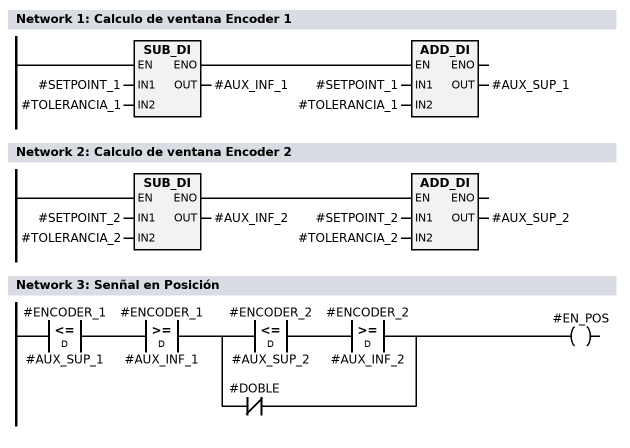
[picture p81: Controlador Posiciones networks 1-3]
NETWORK
TITLE = Calculo de ventana Encoder 1
      A(;
      L     #SETPOINT_1;
      L     #TOLERANCIA_1;
      -D;
      T     #AUX_INF_1;
      AN    OV;
      SAVE;
      CLR;
      A     BR;
      );
      JNB   _001;
      L     #SETPOINT_1;
      L     #TOLERANCIA_1;
      +D;
      T     #AUX_SUP_1;
_001: NOP   0;
NETWORK
TITLE = Calculo de ventana Encoder 2
      A(;
      L     #SETPOINT_2;
      L     #TOLERANCIA_2;
      -D;
      T     #AUX_INF_2;
      AN    OV;
      SAVE;
      CLR;
      A     BR;
      );
      JNB   _002;
      L     #SETPOINT_2;
      L     #TOLERANCIA_2;
      +D;
      T     #AUX_SUP_2;
_002: NOP   0;
NETWORK
TITLE = Senñal en Posición
      A(;
      L     #ENCODER_1;
      L     #AUX_SUP_1;
      <=D;
      );
      A(;
      L     #ENCODER_1;
      L     #AUX_INF_1;
      >=D;
      );
      A(;
      A(;
      L     #ENCODER_2;
      L     #AUX_SUP_2;
      <=D;
      );
      A(;
      L     #ENCODER_2;
      L     #AUX_INF_2;
      >=D;
      );
      ON    #DOBLE;
      );
      =     #EN_POS;
END_FUNCTION

FUNCTION "Almacenes" : VOID	// FC 15
VERSION : 0.1
VAR_TEMP
  TEMP0 : BOOL ;
  TEMP1 : BOOL ;
  TEMP2 : INT ;
END_VAR
BEGIN
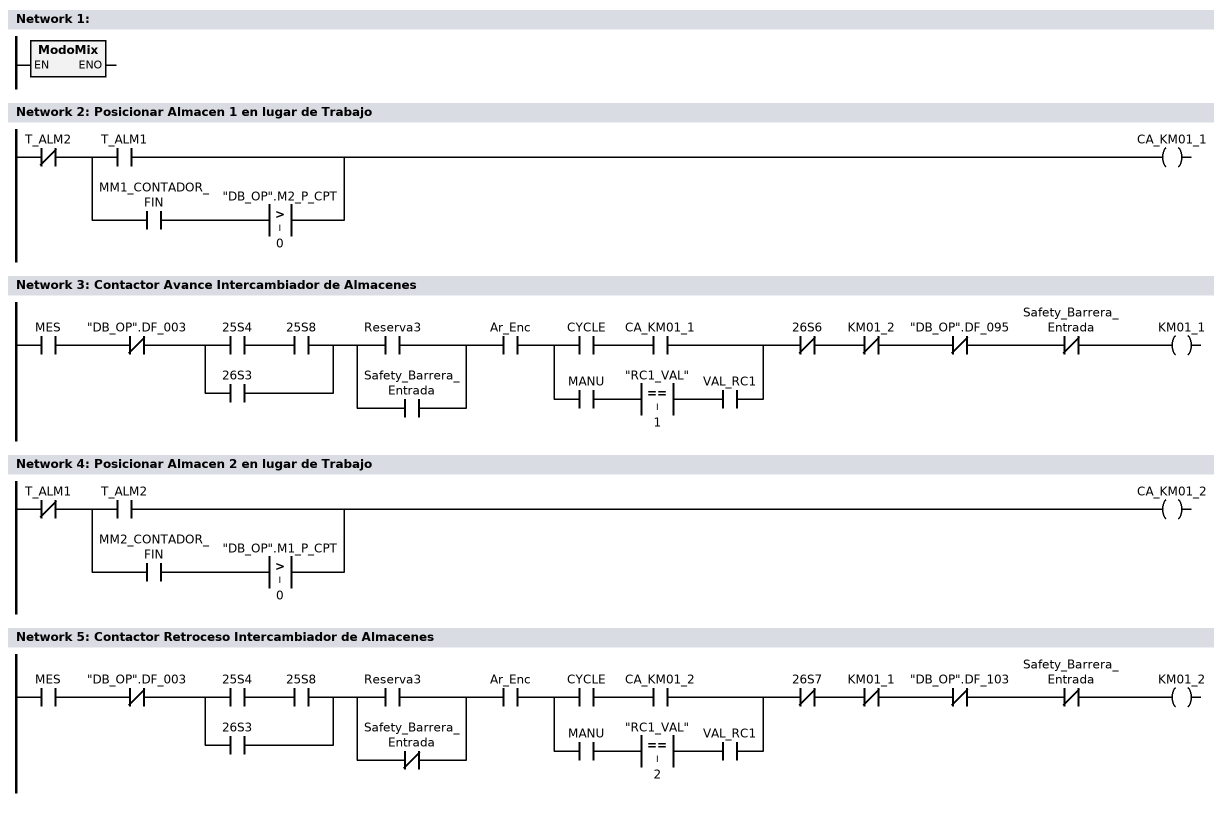
NETWORK
TITLE =
      CALL  "ModoMix";
      NOP   0;
NETWORK
TITLE = Posicionar Almacen 1 en lugar de Trabajo
      AN    "T_ALM2";
      A(;
      O     "T_ALM1";
      O;
      A     "MM1_CONTADOR_FIN";
      A(;
      L     "DB_OP".M2_P_CPT;
      L     0;
      >I;
      );
      );
      =     "CA_KM01_1";
NETWORK
TITLE = Contactor Avance Intercambiador de Almacenes
      A     "MES";
      AN    "DB_OP".DF_003;
      A(;
      A     "25S4";
      A     "25S8";
      O     "26S3";
      );
      A(;
      O     "Reserva3";
      O     "Safety_Barrera_Entrada";
      );
      A     "Ar_Enc";
      A(;
      A     "CYCLE";
      A     "CA_KM01_1";
      O;
      A     "MANU";
      A(;
      L     "RC1_VAL";
      L     1;
      ==I;
      );
      A     "VAL_RC1";
      );
      AN    "26S6";
      AN    "KM01_2";
      AN    "DB_OP".DF_095;
      AN    "Safety_Barrera_Entrada";
      =     "KM01_1";
NETWORK
TITLE = Posicionar Almacen 2 en lugar de Trabajo
      AN    "T_ALM1";
      A(;
      O     "T_ALM2";
      O;
      A     "MM2_CONTADOR_FIN";
      A(;
      L     "DB_OP".M1_P_CPT;
      L     0;
      >I;
      );
      );
      =     "CA_KM01_2";
NETWORK
TITLE = Contactor Retroceso Intercambiador de Almacenes
      A     "MES";
      AN    "DB_OP".DF_003;
      A(;
      A     "25S4";
      A     "25S8";
      O     "26S3";
      );
      A(;
      O     "Reserva3";
      ON    "Safety_Barrera_Entrada";
      );
      A     "Ar_Enc";
      A(;
      A     "CYCLE";
      A     "CA_KM01_2";
      O;
      A     "MANU";
      A(;
      L     "RC1_VAL";
      L     2;
      ==I;
      );
      A     "VAL_RC1";
      );
      AN    "26S7";
      AN    "KM01_1";
      AN    "DB_OP".DF_103;
      AN    "Safety_Barrera_Entrada";
      =     "KM01_2";
END_FUNCTION

FUNCTION "Registro_pos_Plegador" : VOID	// FC 17
TITLE = Registro de posiciones del Plegador
//para verificar el posicionamiento desde el panel
NAME : eProC
VERSION : 0.1
BEGIN
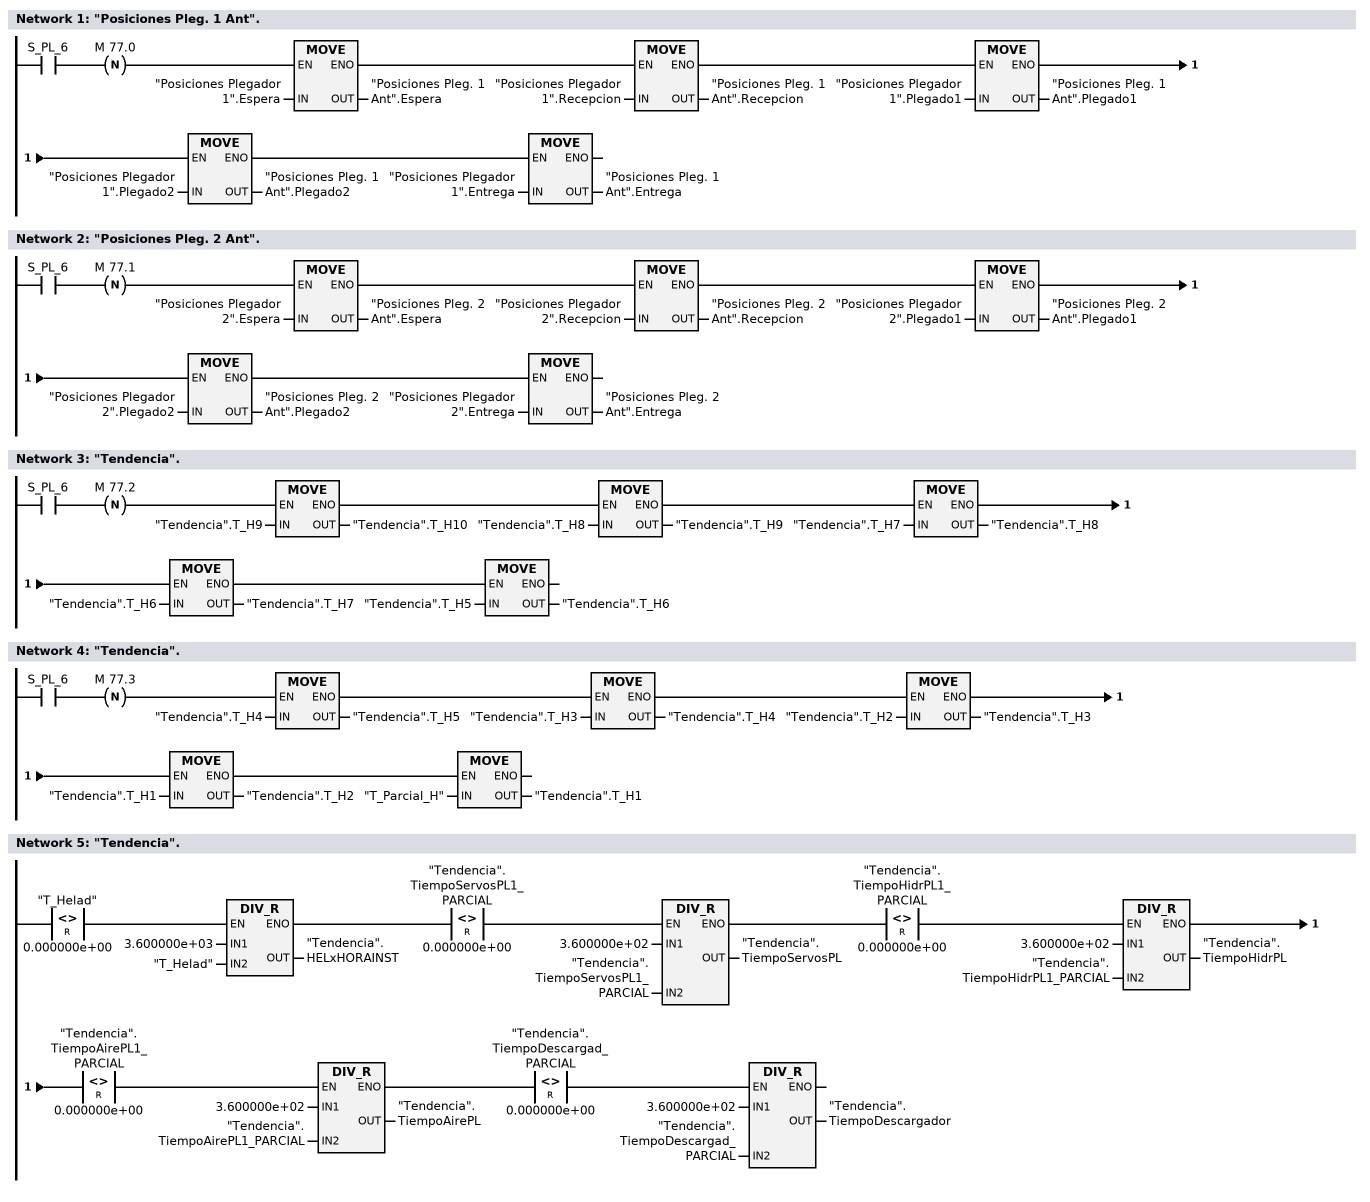
NETWORK
TITLE = "Posiciones Pleg. 1 Ant".
      A(;
      A(;
      A(;
      A(;
      A     "S_PL_6";
      FN    M 77.0;
      JNB   _001;
      L     "Posiciones Plegador 1".Espera;
      T     "Posiciones Pleg. 1 Ant".Espera;
      SET;
      SAVE;
      CLR;
_001: A     BR;
      );
      JNB   _002;
      L     "Posiciones Plegador 1".Recepcion;
      T     "Posiciones Pleg. 1 Ant".Recepcion;
      SET;
      SAVE;
      CLR;
_002: A     BR;
      );
      JNB   _003;
      L     "Posiciones Plegador 1".Plegado1;
      T     "Posiciones Pleg. 1 Ant".Plegado1;
      SET;
      SAVE;
      CLR;
_003: A     BR;
      );
      JNB   _004;
      L     "Posiciones Plegador 1".Plegado2;
      T     "Posiciones Pleg. 1 Ant".Plegado2;
      SET;
      SAVE;
      CLR;
_004: A     BR;
      );
      JNB   _005;
      L     "Posiciones Plegador 1".Entrega;
      T     "Posiciones Pleg. 1 Ant".Entrega;
_005: NOP   0;
NETWORK
TITLE = "Posiciones Pleg. 2 Ant".
      A(;
      A(;
      A(;
      A(;
      A     "S_PL_6";
      FN    M 77.1;
      JNB   _006;
      L     "Posiciones Plegador 2".Espera;
      T     "Posiciones Pleg. 2 Ant".Espera;
      SET;
      SAVE;
      CLR;
_006: A     BR;
      );
      JNB   _007;
      L     "Posiciones Plegador 2".Recepcion;
      T     "Posiciones Pleg. 2 Ant".Recepcion;
      SET;
      SAVE;
      CLR;
_007: A     BR;
      );
      JNB   _008;
      L     "Posiciones Plegador 2".Plegado1;
      T     "Posiciones Pleg. 2 Ant".Plegado1;
      SET;
      SAVE;
      CLR;
_008: A     BR;
      );
      JNB   _009;
      L     "Posiciones Plegador 2".Plegado2;
      T     "Posiciones Pleg. 2 Ant".Plegado2;
      SET;
      SAVE;
      CLR;
_009: A     BR;
      );
      JNB   _00a;
      L     "Posiciones Plegador 2".Entrega;
      T     "Posiciones Pleg. 2 Ant".Entrega;
_00a: NOP   0;
NETWORK
TITLE = "Tendencia".
      A(;
      A(;
      A(;
      A(;
      A     "S_PL_6";
      FN    M 77.2;
      JNB   _00b;
      L     "Tendencia".T_H9;
      T     "Tendencia".T_H10;
      SET;
      SAVE;
      CLR;
_00b: A     BR;
      );
      JNB   _00c;
      L     "Tendencia".T_H8;
      T     "Tendencia".T_H9;
      SET;
      SAVE;
      CLR;
_00c: A     BR;
      );
      JNB   _00d;
      L     "Tendencia".T_H7;
      T     "Tendencia".T_H8;
      SET;
      SAVE;
      CLR;
_00d: A     BR;
      );
      JNB   _00e;
      L     "Tendencia".T_H6;
      T     "Tendencia".T_H7;
      SET;
      SAVE;
      CLR;
_00e: A     BR;
      );
      JNB   _00f;
      L     "Tendencia".T_H5;
      T     "Tendencia".T_H6;
_00f: NOP   0;
NETWORK
TITLE = "Tendencia".
      A(;
      A(;
      A(;
      A(;
      A     "S_PL_6";
      FN    M 77.3;
      JNB   _010;
      L     "Tendencia".T_H4;
      T     "Tendencia".T_H5;
      SET;
      SAVE;
      CLR;
_010: A     BR;
      );
      JNB   _011;
      L     "Tendencia".T_H3;
      T     "Tendencia".T_H4;
      SET;
      SAVE;
      CLR;
_011: A     BR;
      );
      JNB   _012;
      L     "Tendencia".T_H2;
      T     "Tendencia".T_H3;
      SET;
      SAVE;
      CLR;
_012: A     BR;
      );
      JNB   _013;
      L     "Tendencia".T_H1;
      T     "Tendencia".T_H2;
      SET;
      SAVE;
      CLR;
_013: A     BR;
      );
      JNB   _014;
      L     "T_Parcial_H";
      T     "Tendencia".T_H1;
_014: NOP   0;
NETWORK
TITLE = "Tendencia".
      A(;
      A(;
      A(;
      A(;
      A(;
      L     "T_Helad";
      L     0.000000e+00;
      <>R;
      );
      JNB   _015;
      L     3.600000e+03;
      L     "T_Helad";
      /R;
      T     "Tendencia".HELxHORAINST;
      AN    OV;
      SAVE;
      CLR;
_015: A     BR;
      );
      A(;
      L     "Tendencia".TiempoServosPL1_PARCIAL;
      L     0.000000e+00;
      <>R;
      );
      JNB   _016;
      L     3.600000e+02;
      L     "Tendencia".TiempoServosPL1_PARCIAL;
      /R;
      T     "Tendencia".TiempoServosPL;
      AN    OV;
      SAVE;
      CLR;
_016: A     BR;
      );
      A(;
      L     "Tendencia".TiempoHidrPL1_PARCIAL;
      L     0.000000e+00;
      <>R;
      );
      JNB   _017;
      L     3.600000e+02;
      L     "Tendencia".TiempoHidrPL1_PARCIAL;
      /R;
      T     "Tendencia".TiempoHidrPL;
      AN    OV;
      SAVE;
      CLR;
_017: A     BR;
      );
      A(;
      L     "Tendencia".TiempoAirePL1_PARCIAL;
      L     0.000000e+00;
      <>R;
      );
      JNB   _018;
      L     3.600000e+02;
      L     "Tendencia".TiempoAirePL1_PARCIAL;
      /R;
      T     "Tendencia".TiempoAirePL;
      AN    OV;
      SAVE;
      CLR;
_018: A     BR;
      );
      A(;
      L     "Tendencia".TiempoDescargad_PARCIAL;
      L     0.000000e+00;
      <>R;
      );
      JNB   _019;
      L     3.600000e+02;
      L     "Tendencia".TiempoDescargad_PARCIAL;
      /R;
      T     "Tendencia".TiempoDescargador;
_019: NOP   0;
END_FUNCTION

FUNCTION "Registro_pos_Pinza" : VOID	// FC 18
TITLE = Registro de posiciones de la Pinza
//para verificar el posicionamiento desde el panel
NAME : eProC
VERSION : 0.1
BEGIN
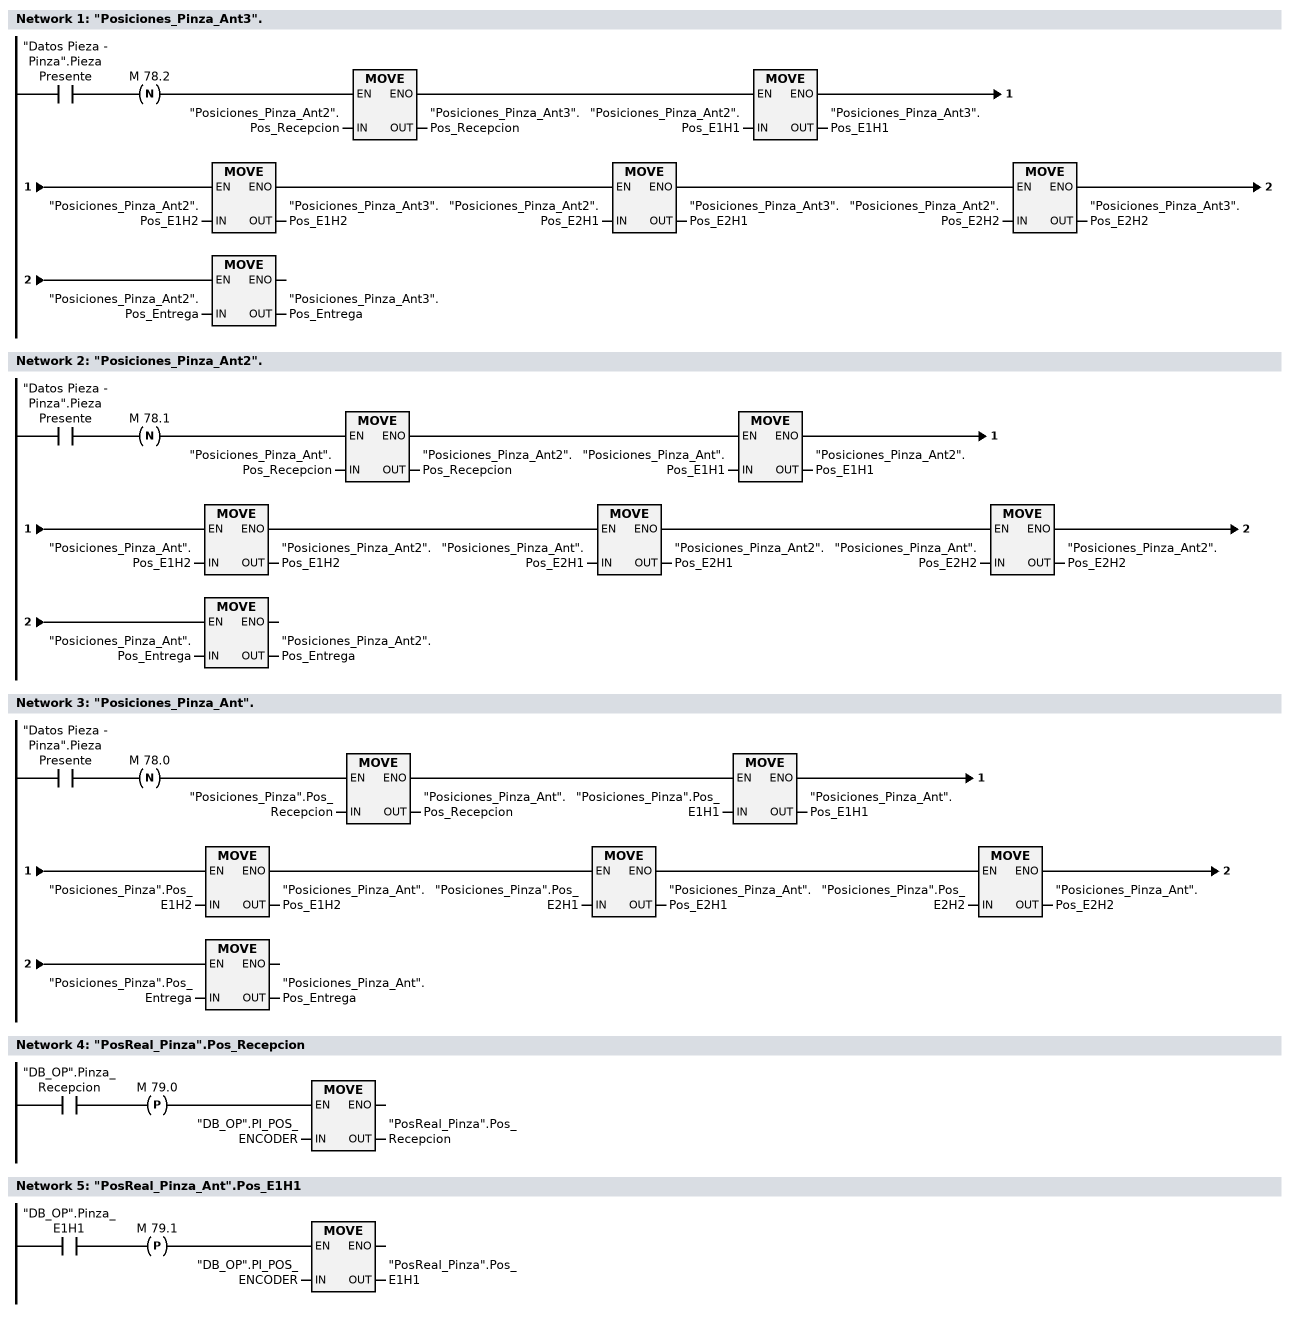
NETWORK
TITLE = "Posiciones_Pinza_Ant3".
      A(;
      A(;
      A(;
      A(;
      A(;
      A     "Datos Pieza - Pinza".PiezaPresente;
      FN    M 78.2;
      JNB   _001;
      L     "Posiciones_Pinza_Ant2".Pos_Recepcion;
      T     "Posiciones_Pinza_Ant3".Pos_Recepcion;
      SET;
      SAVE;
      CLR;
_001: A     BR;
      );
      JNB   _002;
      L     "Posiciones_Pinza_Ant2".Pos_E1H1;
      T     "Posiciones_Pinza_Ant3".Pos_E1H1;
      SET;
      SAVE;
      CLR;
_002: A     BR;
      );
      JNB   _003;
      L     "Posiciones_Pinza_Ant2".Pos_E1H2;
      T     "Posiciones_Pinza_Ant3".Pos_E1H2;
      SET;
      SAVE;
      CLR;
_003: A     BR;
      );
      JNB   _004;
      L     "Posiciones_Pinza_Ant2".Pos_E2H1;
      T     "Posiciones_Pinza_Ant3".Pos_E2H1;
      SET;
      SAVE;
      CLR;
_004: A     BR;
      );
      JNB   _005;
      L     "Posiciones_Pinza_Ant2".Pos_E2H2;
      T     "Posiciones_Pinza_Ant3".Pos_E2H2;
      SET;
      SAVE;
      CLR;
_005: A     BR;
      );
      JNB   _006;
      L     "Posiciones_Pinza_Ant2".Pos_Entrega;
      T     "Posiciones_Pinza_Ant3".Pos_Entrega;
_006: NOP   0;
NETWORK
TITLE = "Posiciones_Pinza_Ant2".
      A(;
      A(;
      A(;
      A(;
      A(;
      A     "Datos Pieza - Pinza".PiezaPresente;
      FN    M 78.1;
      JNB   _007;
      L     "Posiciones_Pinza_Ant".Pos_Recepcion;
      T     "Posiciones_Pinza_Ant2".Pos_Recepcion;
      SET;
      SAVE;
      CLR;
_007: A     BR;
      );
      JNB   _008;
      L     "Posiciones_Pinza_Ant".Pos_E1H1;
      T     "Posiciones_Pinza_Ant2".Pos_E1H1;
      SET;
      SAVE;
      CLR;
_008: A     BR;
      );
      JNB   _009;
      L     "Posiciones_Pinza_Ant".Pos_E1H2;
      T     "Posiciones_Pinza_Ant2".Pos_E1H2;
      SET;
      SAVE;
      CLR;
_009: A     BR;
      );
      JNB   _00a;
      L     "Posiciones_Pinza_Ant".Pos_E2H1;
      T     "Posiciones_Pinza_Ant2".Pos_E2H1;
      SET;
      SAVE;
      CLR;
_00a: A     BR;
      );
      JNB   _00b;
      L     "Posiciones_Pinza_Ant".Pos_E2H2;
      T     "Posiciones_Pinza_Ant2".Pos_E2H2;
      SET;
      SAVE;
      CLR;
_00b: A     BR;
      );
      JNB   _00c;
      L     "Posiciones_Pinza_Ant".Pos_Entrega;
      T     "Posiciones_Pinza_Ant2".Pos_Entrega;
_00c: NOP   0;
NETWORK
TITLE = "Posiciones_Pinza_Ant".
      A(;
      A(;
      A(;
      A(;
      A(;
      A     "Datos Pieza - Pinza".PiezaPresente;
      FN    M 78.0;
      JNB   _00d;
      L     "Posiciones_Pinza".Pos_Recepcion;
      T     "Posiciones_Pinza_Ant".Pos_Recepcion;
      SET;
      SAVE;
      CLR;
_00d: A     BR;
      );
      JNB   _00e;
      L     "Posiciones_Pinza".Pos_E1H1;
      T     "Posiciones_Pinza_Ant".Pos_E1H1;
      SET;
      SAVE;
      CLR;
_00e: A     BR;
      );
      JNB   _00f;
      L     "Posiciones_Pinza".Pos_E1H2;
      T     "Posiciones_Pinza_Ant".Pos_E1H2;
      SET;
      SAVE;
      CLR;
_00f: A     BR;
      );
      JNB   _010;
      L     "Posiciones_Pinza".Pos_E2H1;
      T     "Posiciones_Pinza_Ant".Pos_E2H1;
      SET;
      SAVE;
      CLR;
_010: A     BR;
      );
      JNB   _011;
      L     "Posiciones_Pinza".Pos_E2H2;
      T     "Posiciones_Pinza_Ant".Pos_E2H2;
      SET;
      SAVE;
      CLR;
_011: A     BR;
      );
      JNB   _012;
      L     "Posiciones_Pinza".Pos_Entrega;
      T     "Posiciones_Pinza_Ant".Pos_Entrega;
_012: NOP   0;
NETWORK
TITLE = "PosReal_Pinza".Pos_Recepcion
      A     "DB_OP".Pinza_Recepcion;
      FP    M 79.0;
      JNB   _013;
      L     "DB_OP".PI_POS_ENCODER;
      T     "PosReal_Pinza".Pos_Recepcion;
_013: NOP   0;
NETWORK
TITLE = "PosReal_Pinza_Ant".Pos_E1H1
      A     "DB_OP".Pinza_E1H1;
      FP    M 79.1;
      JNB   _014;
      L     "DB_OP".PI_POS_ENCODER;
      T     "PosReal_Pinza".Pos_E1H1;
_014: NOP   0;
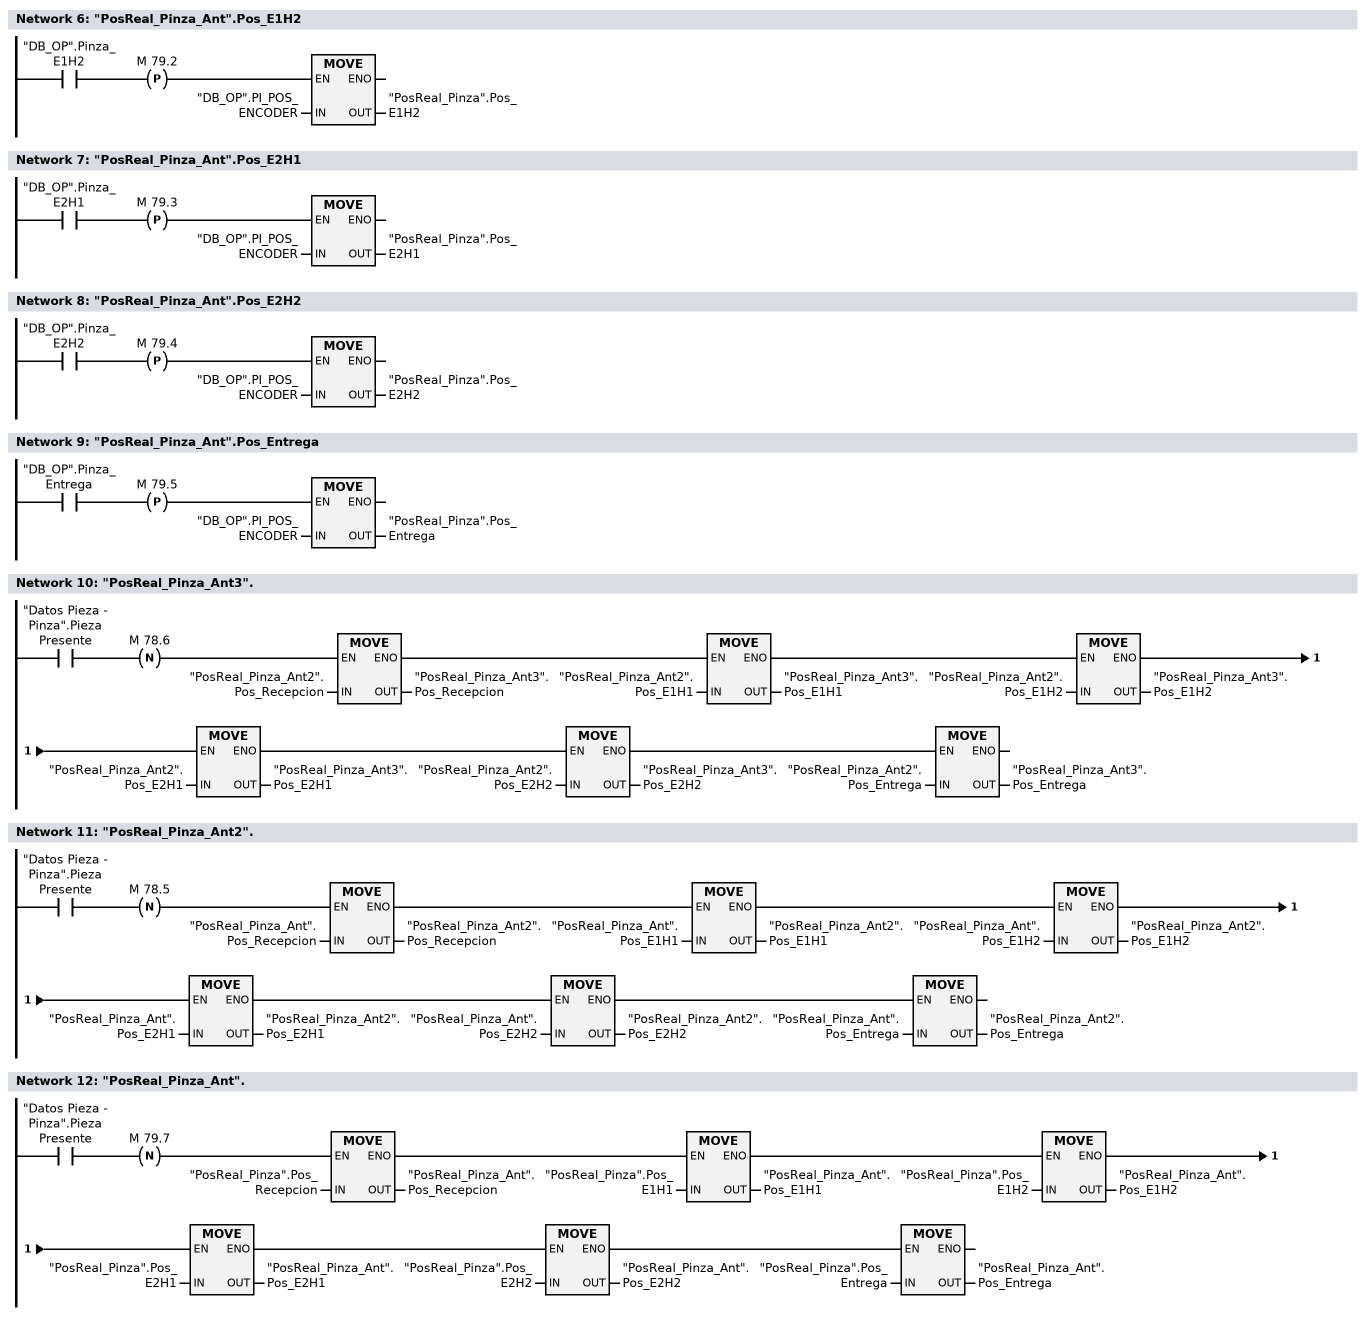
NETWORK
TITLE = "PosReal_Pinza_Ant".Pos_E1H2
      A     "DB_OP".Pinza_E1H2;
      FP    M 79.2;
      JNB   _015;
      L     "DB_OP".PI_POS_ENCODER;
      T     "PosReal_Pinza".Pos_E1H2;
_015: NOP   0;
NETWORK
TITLE = "PosReal_Pinza_Ant".Pos_E2H1
      A     "DB_OP".Pinza_E2H1;
      FP    M 79.3;
      JNB   _016;
      L     "DB_OP".PI_POS_ENCODER;
      T     "PosReal_Pinza".Pos_E2H1;
_016: NOP   0;
NETWORK
TITLE = "PosReal_Pinza_Ant".Pos_E2H2
      A     "DB_OP".Pinza_E2H2;
      FP    M 79.4;
      JNB   _017;
      L     "DB_OP".PI_POS_ENCODER;
      T     "PosReal_Pinza".Pos_E2H2;
_017: NOP   0;
NETWORK
TITLE = "PosReal_Pinza_Ant".Pos_Entrega
      A     "DB_OP".Pinza_Entrega;
      FP    M 79.5;
      JNB   _018;
      L     "DB_OP".PI_POS_ENCODER;
      T     "PosReal_Pinza".Pos_Entrega;
_018: NOP   0;
NETWORK
TITLE = "PosReal_Pinza_Ant3".
      A(;
      A(;
      A(;
      A(;
      A(;
      A     "Datos Pieza - Pinza".PiezaPresente;
      FN    M 78.6;
      JNB   _019;
      L     "PosReal_Pinza_Ant2".Pos_Recepcion;
      T     "PosReal_Pinza_Ant3".Pos_Recepcion;
      SET;
      SAVE;
      CLR;
_019: A     BR;
      );
      JNB   _01a;
      L     "PosReal_Pinza_Ant2".Pos_E1H1;
      T     "PosReal_Pinza_Ant3".Pos_E1H1;
      SET;
      SAVE;
      CLR;
_01a: A     BR;
      );
      JNB   _01b;
      L     "PosReal_Pinza_Ant2".Pos_E1H2;
      T     "PosReal_Pinza_Ant3".Pos_E1H2;
      SET;
      SAVE;
      CLR;
_01b: A     BR;
      );
      JNB   _01c;
      L     "PosReal_Pinza_Ant2".Pos_E2H1;
      T     "PosReal_Pinza_Ant3".Pos_E2H1;
      SET;
      SAVE;
      CLR;
_01c: A     BR;
      );
      JNB   _01d;
      L     "PosReal_Pinza_Ant2".Pos_E2H2;
      T     "PosReal_Pinza_Ant3".Pos_E2H2;
      SET;
      SAVE;
      CLR;
_01d: A     BR;
      );
      JNB   _01e;
      L     "PosReal_Pinza_Ant2".Pos_Entrega;
      T     "PosReal_Pinza_Ant3".Pos_Entrega;
_01e: NOP   0;
NETWORK
TITLE = "PosReal_Pinza_Ant2".
      A(;
      A(;
      A(;
      A(;
      A(;
      A     "Datos Pieza - Pinza".PiezaPresente;
      FN    M 78.5;
      JNB   _01f;
      L     "PosReal_Pinza_Ant".Pos_Recepcion;
      T     "PosReal_Pinza_Ant2".Pos_Recepcion;
      SET;
      SAVE;
      CLR;
_01f: A     BR;
      );
      JNB   _020;
      L     "PosReal_Pinza_Ant".Pos_E1H1;
      T     "PosReal_Pinza_Ant2".Pos_E1H1;
      SET;
      SAVE;
      CLR;
_020: A     BR;
      );
      JNB   _021;
      L     "PosReal_Pinza_Ant".Pos_E1H2;
      T     "PosReal_Pinza_Ant2".Pos_E1H2;
      SET;
      SAVE;
      CLR;
_021: A     BR;
      );
      JNB   _022;
      L     "PosReal_Pinza_Ant".Pos_E2H1;
      T     "PosReal_Pinza_Ant2".Pos_E2H1;
      SET;
      SAVE;
      CLR;
_022: A     BR;
      );
      JNB   _023;
      L     "PosReal_Pinza_Ant".Pos_E2H2;
      T     "PosReal_Pinza_Ant2".Pos_E2H2;
      SET;
      SAVE;
      CLR;
_023: A     BR;
      );
      JNB   _024;
      L     "PosReal_Pinza_Ant".Pos_Entrega;
      T     "PosReal_Pinza_Ant2".Pos_Entrega;
_024: NOP   0;
NETWORK
TITLE = "PosReal_Pinza_Ant".
      A(;
      A(;
      A(;
      A(;
      A(;
      A     "Datos Pieza - Pinza".PiezaPresente;
      FN    M 79.7;
      JNB   _025;
      L     "PosReal_Pinza".Pos_Recepcion;
      T     "PosReal_Pinza_Ant".Pos_Recepcion;
      SET;
      SAVE;
      CLR;
_025: A     BR;
      );
      JNB   _026;
      L     "PosReal_Pinza".Pos_E1H1;
      T     "PosReal_Pinza_Ant".Pos_E1H1;
      SET;
      SAVE;
      CLR;
_026: A     BR;
      );
      JNB   _027;
      L     "PosReal_Pinza".Pos_E1H2;
      T     "PosReal_Pinza_Ant".Pos_E1H2;
      SET;
      SAVE;
      CLR;
_027: A     BR;
      );
      JNB   _028;
      L     "PosReal_Pinza".Pos_E2H1;
      T     "PosReal_Pinza_Ant".Pos_E2H1;
      SET;
      SAVE;
      CLR;
_028: A     BR;
      );
      JNB   _029;
      L     "PosReal_Pinza".Pos_E2H2;
      T     "PosReal_Pinza_Ant".Pos_E2H2;
      SET;
      SAVE;
      CLR;
_029: A     BR;
      );
      JNB   _02a;
      L     "PosReal_Pinza".Pos_Entrega;
      T     "PosReal_Pinza_Ant".Pos_Entrega;
_02a: NOP   0;
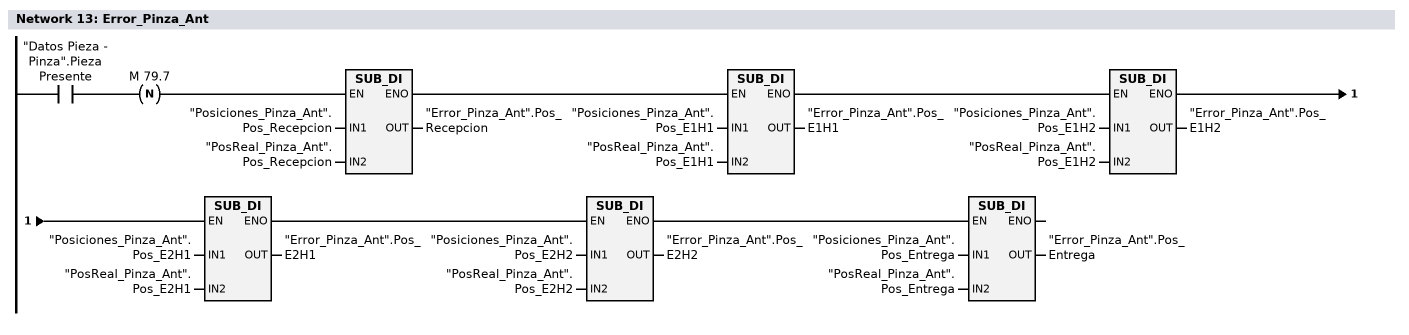
NETWORK
TITLE = Error_Pinza_Ant
      A(;
      A(;
      A(;
      A(;
      A(;
      A     "Datos Pieza - Pinza".PiezaPresente;
      FN    M 79.7;
      JNB   _02b;
      L     "Posiciones_Pinza_Ant".Pos_Recepcion;
      L     "PosReal_Pinza_Ant".Pos_Recepcion;
      -D;
      T     "Error_Pinza_Ant".Pos_Recepcion;
      AN    OV;
      SAVE;
      CLR;
_02b: A     BR;
      );
      JNB   _02c;
      L     "Posiciones_Pinza_Ant".Pos_E1H1;
      L     "PosReal_Pinza_Ant".Pos_E1H1;
      -D;
      T     "Error_Pinza_Ant".Pos_E1H1;
      AN    OV;
      SAVE;
      CLR;
_02c: A     BR;
      );
      JNB   _02d;
      L     "Posiciones_Pinza_Ant".Pos_E1H2;
      L     "PosReal_Pinza_Ant".Pos_E1H2;
      -D;
      T     "Error_Pinza_Ant".Pos_E1H2;
      AN    OV;
      SAVE;
      CLR;
_02d: A     BR;
      );
      JNB   _02e;
      L     "Posiciones_Pinza_Ant".Pos_E2H1;
      L     "PosReal_Pinza_Ant".Pos_E2H1;
      -D;
      T     "Error_Pinza_Ant".Pos_E2H1;
      AN    OV;
      SAVE;
      CLR;
_02e: A     BR;
      );
      JNB   _02f;
      L     "Posiciones_Pinza_Ant".Pos_E2H2;
      L     "PosReal_Pinza_Ant".Pos_E2H2;
      -D;
      T     "Error_Pinza_Ant".Pos_E2H2;
      AN    OV;
      SAVE;
      CLR;
_02f: A     BR;
      );
      JNB   _030;
      L     "Posiciones_Pinza_Ant".Pos_Entrega;
      L     "PosReal_Pinza_Ant".Pos_Entrega;
      -D;
      T     "Error_Pinza_Ant".Pos_Entrega;
_030: NOP   0;
END_FUNCTION

FUNCTION "Araña" : VOID	// FC 20
VERSION : 0.1
VAR_TEMP
  AUX_VELOCIDAD : INT ;	//Auxiliar Consigna de Velocidad
  AUX_CHAPA_COMPLETA : DINT ;
  Arana_A : DINT ;
  Arana_C : DINT ;
  Arana_D : DINT ;
END_VAR
BEGIN
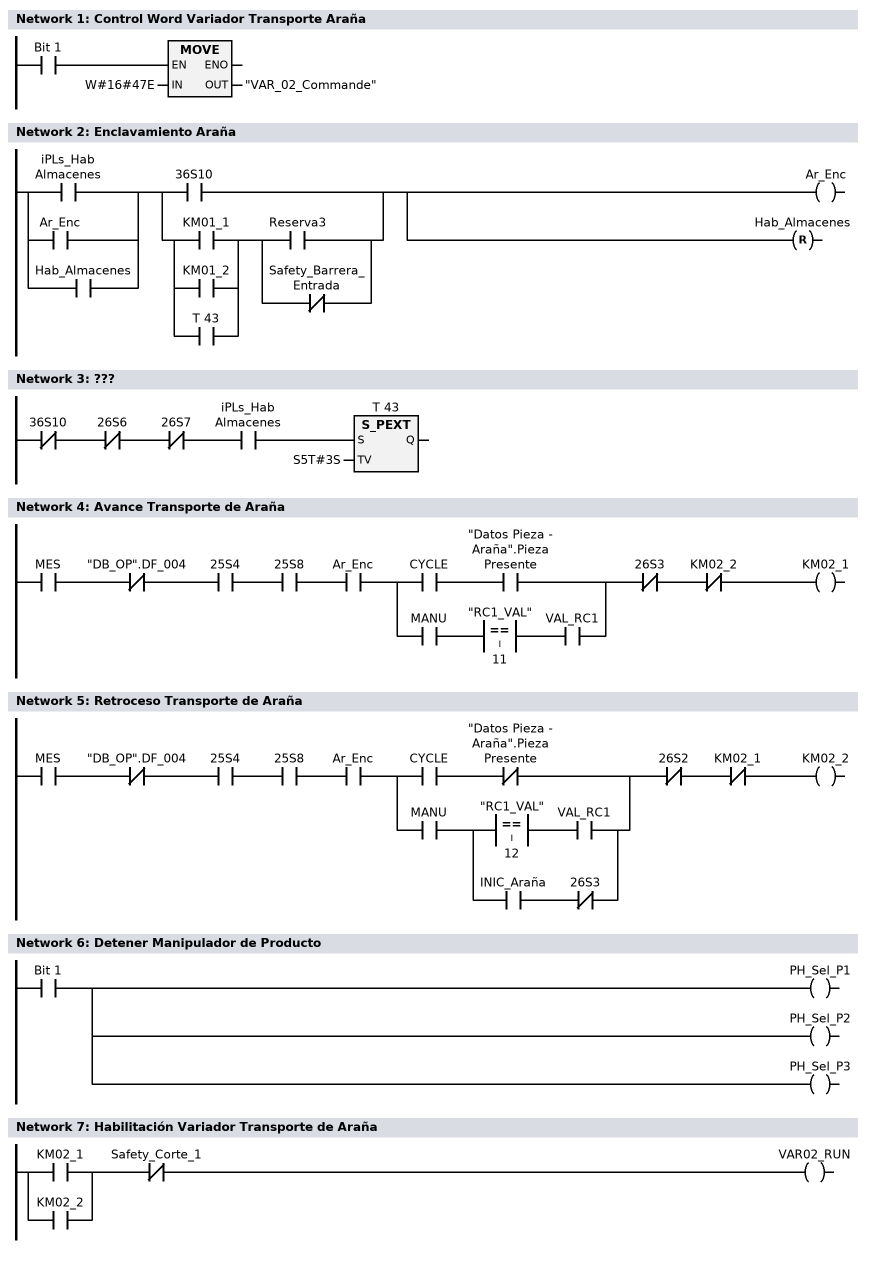
NETWORK
TITLE = Control Word Variador Transporte Araña
      A     "Bit 1";
      JNB   _001;
      L     W#16#47E;
      T     "VAR_02_Commande";
_001: NOP   0;
NETWORK
TITLE = Enclavamiento Araña
      A(;
      O     "iPLs_HabAlmacenes";
      O     "Ar_Enc";
      O     "Hab_Almacenes";
      );
      A(;
      O     "36S10";
      O;
      A(;
      O     "KM01_1";
      O     "KM01_2";
      O     T 43;
      );
      A(;
      O     "Reserva3";
      ON    "Safety_Barrera_Entrada";
      );
      );
      =     "Ar_Enc";
      R     "Hab_Almacenes";
NETWORK
TITLE = ???
      AN    "36S10";
      AN    "26S6";
      AN    "26S7";
      A     "iPLs_HabAlmacenes";
      L     S5T#3S;
      SE    T 43;
      NOP   0;
      NOP   0;
      NOP   0;
      NOP   0;
NETWORK
TITLE = Avance Transporte de Araña
      A     "MES";
      AN    "DB_OP".DF_004;
      A     "25S4";
      A     "25S8";
      A     "Ar_Enc";
      A(;
      A     "CYCLE";
      A     "Datos Pieza - Araña".PiezaPresente;
      O;
      A     "MANU";
      A(;
      L     "RC1_VAL";
      L     11;
      ==I;
      );
      A     "VAL_RC1";
      );
      AN    "26S3";
      AN    "KM02_2";
      =     "KM02_1";
NETWORK
TITLE = Retroceso Transporte de Araña
      A     "MES";
      AN    "DB_OP".DF_004;
      A     "25S4";
      A     "25S8";
      A     "Ar_Enc";
      A(;
      A     "CYCLE";
      AN    "Datos Pieza - Araña".PiezaPresente;
      O;
      A     "MANU";
      A(;
      A(;
      L     "RC1_VAL";
      L     12;
      ==I;
      );
      A     "VAL_RC1";
      O;
      A     "INIC_Araña";
      AN    "26S3";
      );
      );
      AN    "26S2";
      AN    "KM02_1";
      =     "KM02_2";
NETWORK
TITLE = Detener Manipulador de Producto 
      A     "Bit 1";
      =     "PH_Sel_P1";
      =     "PH_Sel_P2";
      =     "PH_Sel_P3";
NETWORK
TITLE = Habilitación Variador Transporte de Araña
      A(;
      O     "KM02_1";
      O     "KM02_2";
      );
      AN    "Safety_Corte_1";
      =     "VAR02_RUN";
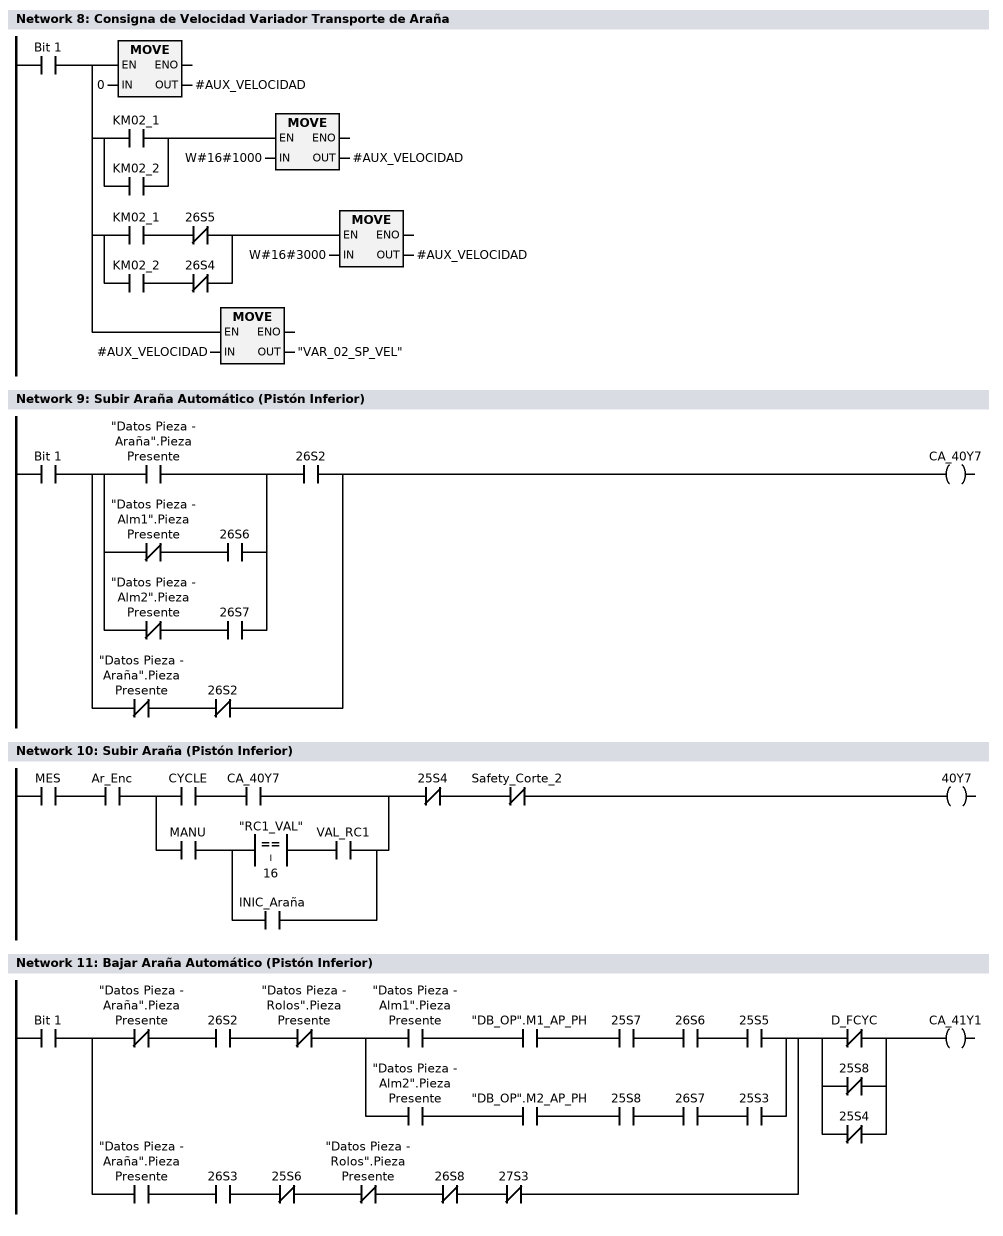
NETWORK
TITLE = Consigna de Velocidad Variador Transporte de Araña
      A     "Bit 1";
      =     L 18.0;
      A     L 18.0;
      JNB   _002;
      L     0;
      T     #AUX_VELOCIDAD;
_002: NOP   0;
      A     L 18.0;
      A(;
      O     "KM02_1";
      O     "KM02_2";
      );
      JNB   _003;
      L     W#16#1000;
      T     #AUX_VELOCIDAD;
_003: NOP   0;
      A     L 18.0;
      A(;
      A     "KM02_1";
      AN    "26S5";
      O;
      A     "KM02_2";
      AN    "26S4";
      );
      JNB   _004;
      L     W#16#3000;
      T     #AUX_VELOCIDAD;
_004: NOP   0;
      A     L 18.0;
      JNB   _005;
      L     #AUX_VELOCIDAD;
      T     "VAR_02_SP_VEL";
_005: NOP   0;
NETWORK
TITLE = Subir Araña Automático (Pistón Inferior)
      A     "Bit 1";
      A(;
      A(;
      O     "Datos Pieza - Araña".PiezaPresente;
      O;
      AN    "Datos Pieza - Alm1".PiezaPresente;
      A     "26S6";
      O;
      AN    "Datos Pieza - Alm2".PiezaPresente;
      A     "26S7";
      );
      A     "26S2";
      O;
      AN    "Datos Pieza - Araña".PiezaPresente;
      AN    "26S2";
      );
      =     "CA_40Y7";
NETWORK
TITLE = Subir Araña (Pistón Inferior)
      A     "MES";
      A     "Ar_Enc";
      A(;
      A     "CYCLE";
      A     "CA_40Y7";
      O;
      A     "MANU";
      A(;
      A(;
      L     "RC1_VAL";
      L     16;
      ==I;
      );
      A     "VAL_RC1";
      O     "INIC_Araña";
      );
      );
      AN    "25S4";
      AN    "Safety_Corte_2";
      =     "40Y7";
NETWORK
TITLE = Bajar Araña Automático (Pistón Inferior)
      A     "Bit 1";
      A(;
      AN    "Datos Pieza - Araña".PiezaPresente;
      A     "26S2";
      AN    "Datos Pieza - Rolos".PiezaPresente;
      A(;
      A     "Datos Pieza - Alm1".PiezaPresente;
      A     "DB_OP".M1_AP_PH;
      A     "25S7";
      A     "26S6";
      A     "25S5";
      O;
      A     "Datos Pieza - Alm2".PiezaPresente;
      A     "DB_OP".M2_AP_PH;
      A     "25S8";
      A     "26S7";
      A     "25S3";
      );
      O;
      A     "Datos Pieza - Araña".PiezaPresente;
      A     "26S3";
      AN    "25S6";
      AN    "Datos Pieza - Rolos".PiezaPresente;
      AN    "26S8";
      AN    "27S3";
      );
      A(;
      ON    "D_FCYC";
      ON    "25S8";
      ON    "25S4";
      );
      =     "CA_41Y1";
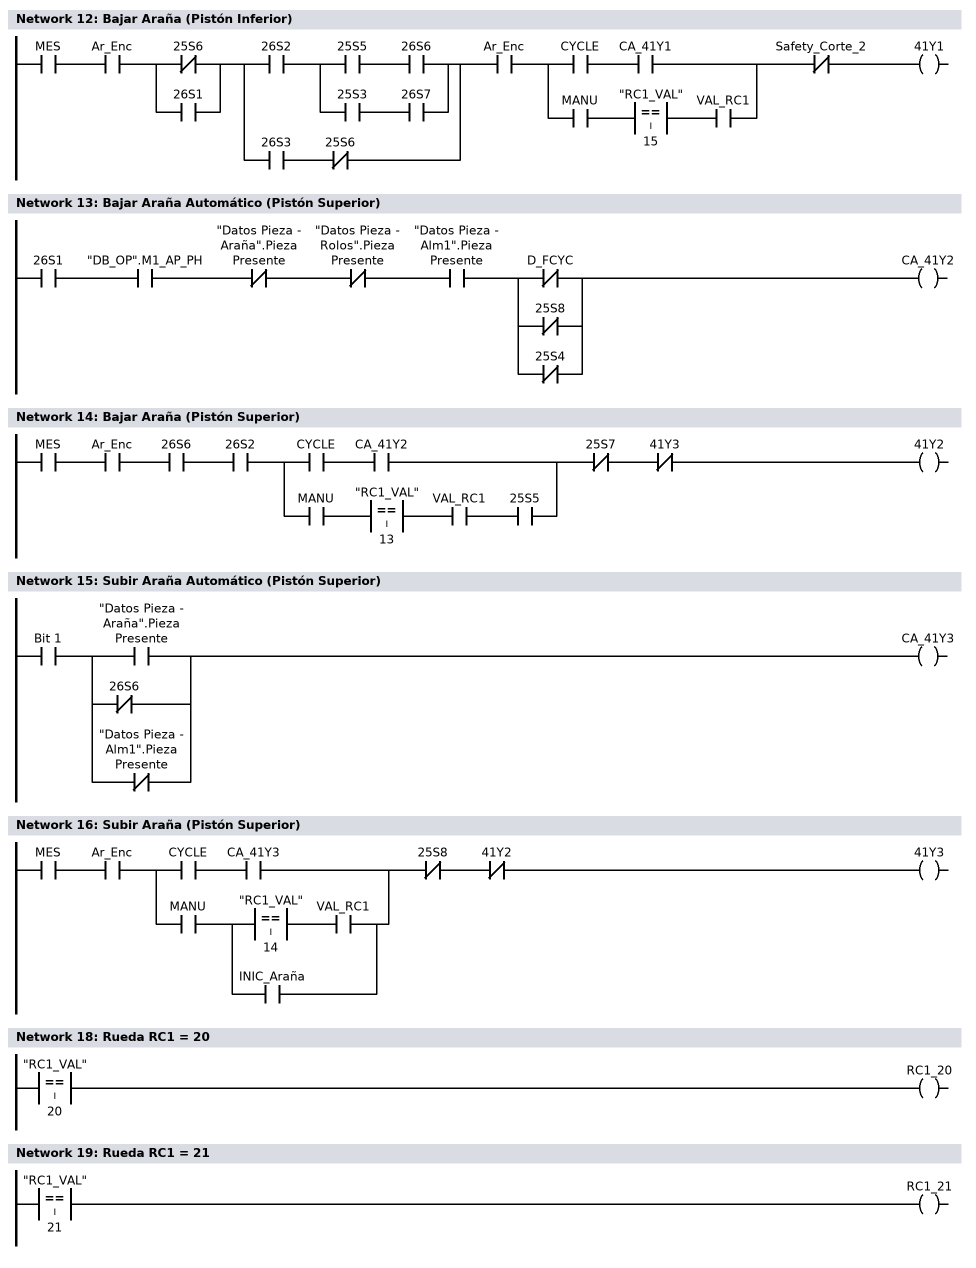
NETWORK
TITLE = Bajar Araña (Pistón Inferior)
      A     "MES";
      A     "Ar_Enc";
      A(;
      ON    "25S6";
      O     "26S1";
      );
      A(;
      A     "26S2";
      A(;
      A     "25S5";
      A     "26S6";
      O;
      A     "25S3";
      A     "26S7";
      );
      O;
      A     "26S3";
      AN    "25S6";
      );
      A     "Ar_Enc";
      A(;
      A     "CYCLE";
      A     "CA_41Y1";
      O;
      A     "MANU";
      A(;
      L     "RC1_VAL";
      L     15;
      ==I;
      );
      A     "VAL_RC1";
      );
      AN    "Safety_Corte_2";
      =     "41Y1";
NETWORK
TITLE = Bajar Araña Automático (Pistón Superior)
      A     "26S1";
      A     "DB_OP".M1_AP_PH;
      AN    "Datos Pieza - Araña".PiezaPresente;
      AN    "Datos Pieza - Rolos".PiezaPresente;
      A     "Datos Pieza - Alm1".PiezaPresente;
      A(;
      ON    "D_FCYC";
      ON    "25S8";
      ON    "25S4";
      );
      =     "CA_41Y2";
NETWORK
TITLE = Bajar Araña (Pistón Superior)
      A     "MES";
      A     "Ar_Enc";
      A     "26S6";
      A     "26S2";
      A(;
      A     "CYCLE";
      A     "CA_41Y2";
      O;
      A     "MANU";
      A(;
      L     "RC1_VAL";
      L     13;
      ==I;
      );
      A     "VAL_RC1";
      A     "25S5";
      );
      AN    "25S7";
      AN    "41Y3";
      =     "41Y2";
NETWORK
TITLE = Subir Araña Automático (Pistón Superior)
      A     "Bit 1";
      A(;
      O     "Datos Pieza - Araña".PiezaPresente;
      ON    "26S6";
      ON    "Datos Pieza - Alm1".PiezaPresente;
      );
      =     "CA_41Y3";
NETWORK
TITLE = Subir Araña (Pistón Superior)
      A     "MES";
      A     "Ar_Enc";
      A(;
      A     "CYCLE";
      A     "CA_41Y3";
      O;
      A     "MANU";
      A(;
      A(;
      L     "RC1_VAL";
      L     14;
      ==I;
      );
      A     "VAL_RC1";
      O     "INIC_Araña";
      );
      );
      AN    "25S8";
      AN    "41Y2";
      =     "41Y3";
NETWORK
TITLE = (COMENTADO EN AWL)
//      U     "MANU"
//      U(    
//      O(    
//      L     "RC1_VAL"
//      L     20
//      ==I   
//      )     
//      O(    
//      L     "RC1_VAL"
//      L     22
//      ==I   
//      )     
//     )     
//      =     #TEMP1
NETWORK
TITLE = Rueda RC1 = 20
      L     "RC1_VAL";
      L     20;
      ==I;
      =     "RC1_20";
NETWORK
TITLE = Rueda RC1 = 21
      L     "RC1_VAL";
      L     21;
      ==I;
      =     "RC1_21";
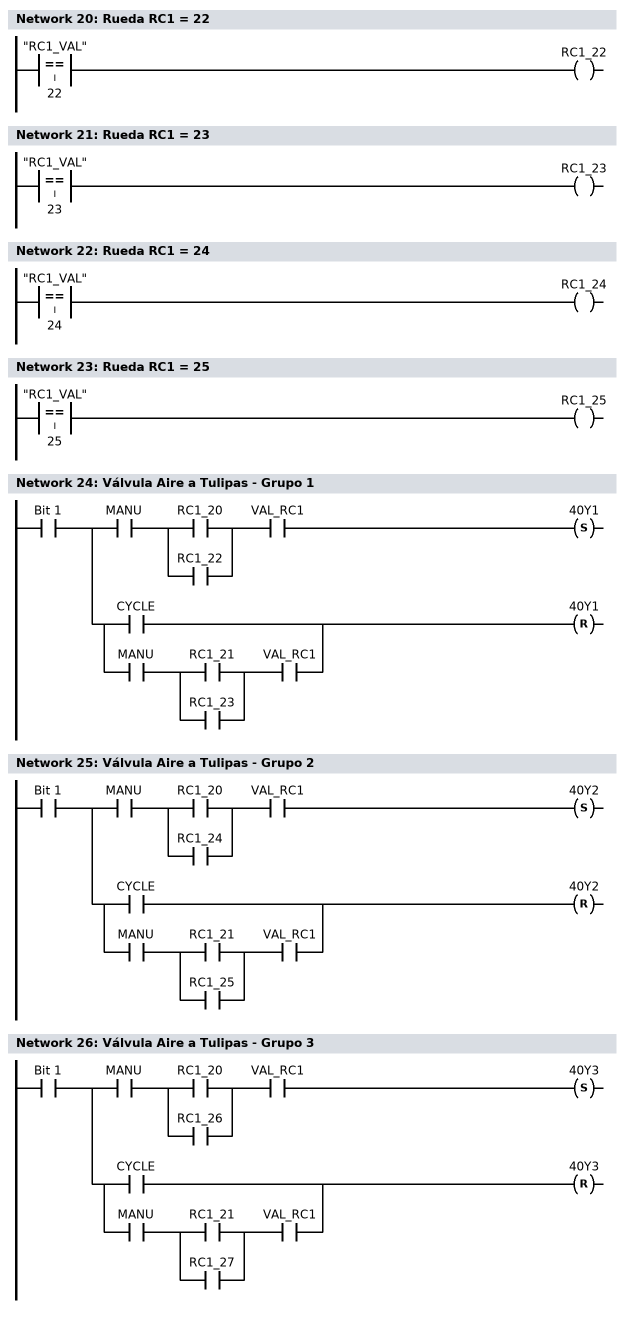
NETWORK
TITLE = Rueda RC1 = 22
      L     "RC1_VAL";
      L     22;
      ==I;
      =     "RC1_22";
NETWORK
TITLE = Rueda RC1 = 23
      L     "RC1_VAL";
      L     23;
      ==I;
      =     "RC1_23";
NETWORK
TITLE = Rueda RC1 = 24
      L     "RC1_VAL";
      L     24;
      ==I;
      =     "RC1_24";
NETWORK
TITLE = Rueda RC1 = 25
      L     "RC1_VAL";
      L     25;
      ==I;
      =     "RC1_25";
NETWORK
TITLE = Válvula Aire a Tulipas - Grupo 1
      A     "Bit 1";
      =     L 18.0;
      A     L 18.0;
      A     "MANU";
      A(;
      O     "RC1_20";
      O     "RC1_22";
      );
      A     "VAL_RC1";
      S     "40Y1";
      A     L 18.0;
      A(;
      O     "CYCLE";
      O;
      A     "MANU";
      A(;
      O     "RC1_21";
      O     "RC1_23";
      );
      A     "VAL_RC1";
      );
      R     "40Y1";
NETWORK
TITLE = Válvula Aire a Tulipas - Grupo 2
      A     "Bit 1";
      =     L 18.0;
      A     L 18.0;
      A     "MANU";
      A(;
      O     "RC1_20";
      O     "RC1_24";
      );
      A     "VAL_RC1";
      S     "40Y2";
      A     L 18.0;
      A(;
      O     "CYCLE";
      O;
      A     "MANU";
      A(;
      O     "RC1_21";
      O     "RC1_25";
      );
      A     "VAL_RC1";
      );
      R     "40Y2";
NETWORK
TITLE = Válvula Aire a Tulipas - Grupo 3
      A     "Bit 1";
      =     L 18.0;
      A     L 18.0;
      A     "MANU";
      A(;
      O     "RC1_20";
      O     "RC1_26";
      );
      A     "VAL_RC1";
      S     "40Y3";
      A     L 18.0;
      A(;
      O     "CYCLE";
      O;
      A     "MANU";
      A(;
      O     "RC1_21";
      O     "RC1_27";
      );
      A     "VAL_RC1";
      );
      R     "40Y3";
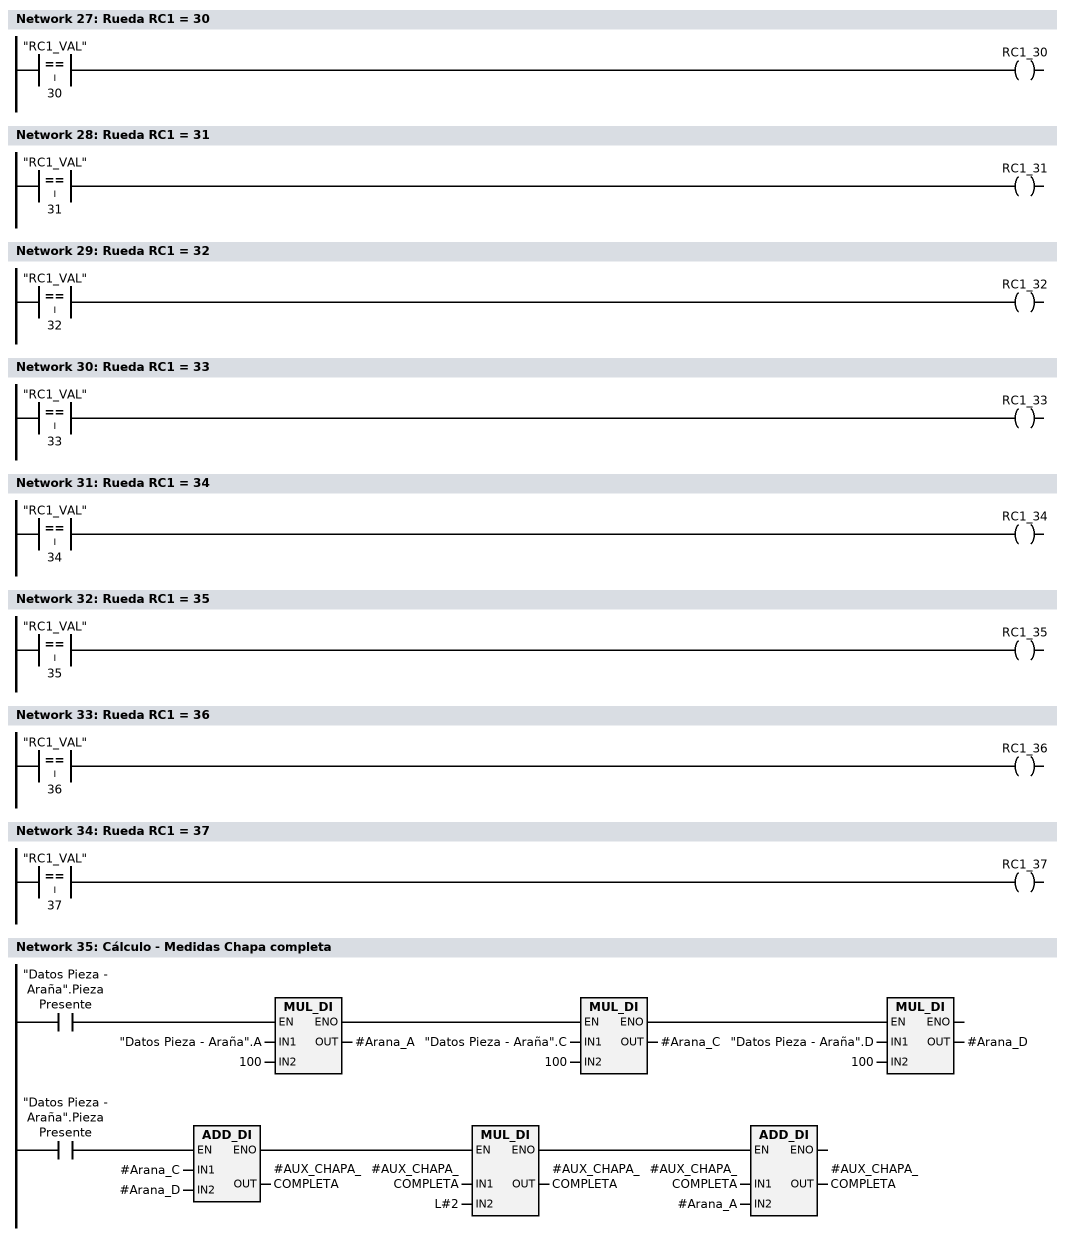
NETWORK
TITLE = Rueda RC1 = 30
      L     "RC1_VAL";
      L     30;
      ==I;
      =     "RC1_30";
NETWORK
TITLE = Rueda RC1 = 31
      L     "RC1_VAL";
      L     31;
      ==I;
      =     "RC1_31";
NETWORK
TITLE = Rueda RC1 = 32
      L     "RC1_VAL";
      L     32;
      ==I;
      =     "RC1_32";
NETWORK
TITLE = Rueda RC1 = 33
      L     "RC1_VAL";
      L     33;
      ==I;
      =     "RC1_33";
NETWORK
TITLE = Rueda RC1 = 34
      L     "RC1_VAL";
      L     34;
      ==I;
      =     "RC1_34";
NETWORK
TITLE = Rueda RC1 = 35
      L     "RC1_VAL";
      L     35;
      ==I;
      =     "RC1_35";
NETWORK
TITLE = Rueda RC1 = 36
      L     "RC1_VAL";
      L     36;
      ==I;
      =     "RC1_36";
NETWORK
TITLE = Rueda RC1 = 37
      L     "RC1_VAL";
      L     37;
      ==I;
      =     "RC1_37";
NETWORK
TITLE = Cálculo - Medidas Chapa completa 
      A     "Datos Pieza - Araña".PiezaPresente;
      =     L 18.0;
      A(;
      A(;
      A     L 18.0;
      JNB   _006;
      L     "Datos Pieza - Araña".A;
      L     100;
      *D;
      T     #Arana_A;
      AN    OV;
      SAVE;
      CLR;
_006: A     BR;
      );
      JNB   _007;
      L     "Datos Pieza - Araña".C;
      L     100;
      *D;
      T     #Arana_C;
      AN    OV;
      SAVE;
      CLR;
_007: A     BR;
      );
      JNB   _008;
      L     "Datos Pieza - Araña".D;
      L     100;
      *D;
      T     #Arana_D;
_008: NOP   0;
      A(;
      A(;
      A     L 18.0;
      JNB   _009;
      L     #Arana_C;
      L     #Arana_D;
      +D;
      T     #AUX_CHAPA_COMPLETA;
      AN    OV;
      SAVE;
      CLR;
_009: A     BR;
      );
      JNB   _00a;
      L     #AUX_CHAPA_COMPLETA;
      L     L#2;
      *D;
      T     #AUX_CHAPA_COMPLETA;
      AN    OV;
      SAVE;
      CLR;
_00a: A     BR;
      );
      JNB   _00b;
      L     #AUX_CHAPA_COMPLETA;
      L     #Arana_A;
      +D;
      T     #AUX_CHAPA_COMPLETA;
_00b: NOP   0;
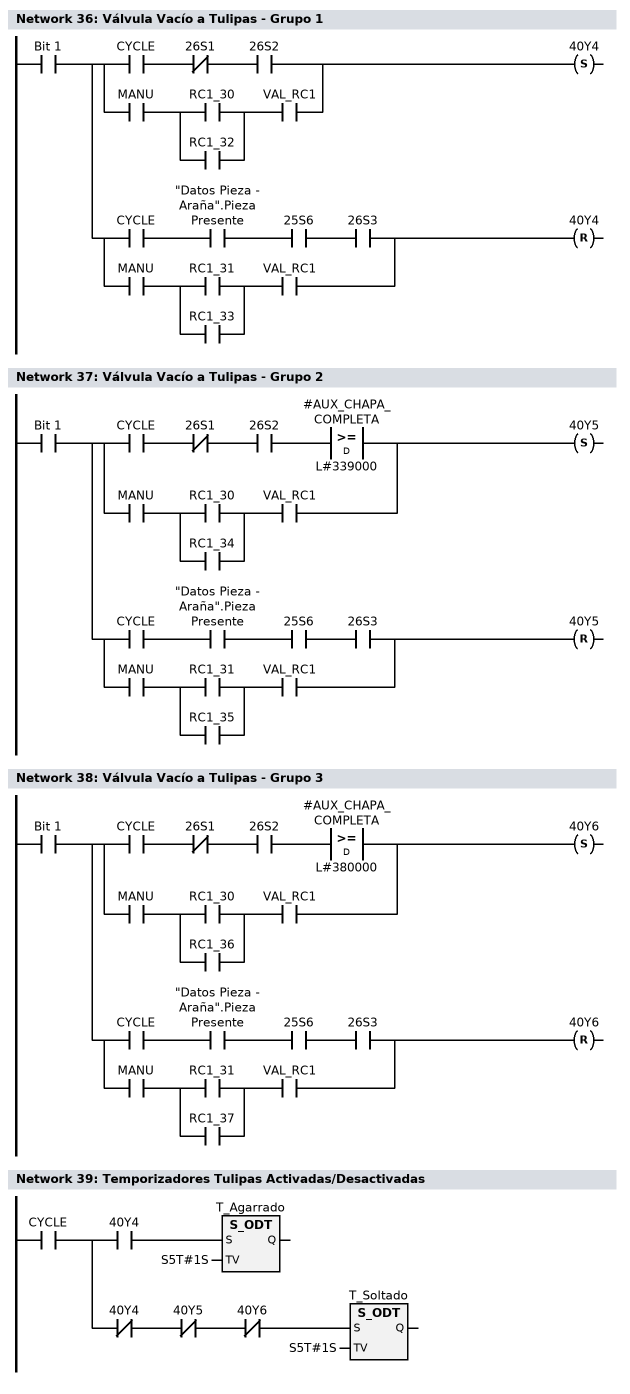
NETWORK
TITLE = Válvula Vacío a Tulipas - Grupo 1
      A     "Bit 1";
      =     L 18.0;
      A     L 18.0;
      A(;
      A     "CYCLE";
      AN    "26S1";
      A     "26S2";
      O;
      A     "MANU";
      A(;
      O     "RC1_30";
      O     "RC1_32";
      );
      A     "VAL_RC1";
      );
      S     "40Y4";
      A     L 18.0;
      A(;
      A     "CYCLE";
      A     "Datos Pieza - Araña".PiezaPresente;
      A     "25S6";
      A     "26S3";
      O;
      A     "MANU";
      A(;
      O     "RC1_31";
      O     "RC1_33";
      );
      A     "VAL_RC1";
      );
      R     "40Y4";
NETWORK
TITLE = Válvula Vacío a Tulipas - Grupo 2
      A     "Bit 1";
      =     L 18.0;
      A     L 18.0;
      A(;
      A     "CYCLE";
      AN    "26S1";
      A     "26S2";
      A(;
      L     #AUX_CHAPA_COMPLETA;
      L     L#339000;
      >=D;
      );
      O;
      A     "MANU";
      A(;
      O     "RC1_30";
      O     "RC1_34";
      );
      A     "VAL_RC1";
      );
      S     "40Y5";
      A     L 18.0;
      A(;
      A     "CYCLE";
      A     "Datos Pieza - Araña".PiezaPresente;
      A     "25S6";
      A     "26S3";
      O;
      A     "MANU";
      A(;
      O     "RC1_31";
      O     "RC1_35";
      );
      A     "VAL_RC1";
      );
      R     "40Y5";
NETWORK
TITLE = Válvula Vacío a Tulipas - Grupo 3
      A     "Bit 1";
      =     L 18.0;
      A     L 18.0;
      A(;
      A     "CYCLE";
      AN    "26S1";
      A     "26S2";
      A(;
      L     #AUX_CHAPA_COMPLETA;
      L     L#380000;
      >=D;
      );
      O;
      A     "MANU";
      A(;
      O     "RC1_30";
      O     "RC1_36";
      );
      A     "VAL_RC1";
      );
      S     "40Y6";
      A     L 18.0;
      A(;
      A     "CYCLE";
      A     "Datos Pieza - Araña".PiezaPresente;
      A     "25S6";
      A     "26S3";
      O;
      A     "MANU";
      A(;
      O     "RC1_31";
      O     "RC1_37";
      );
      A     "VAL_RC1";
      );
      R     "40Y6";
NETWORK
TITLE = Temporizadores Tulipas Activadas/Desactivadas
      A     "CYCLE";
      =     L 18.0;
      A     L 18.0;
      A     "40Y4";
      L     S5T#1S;
      SD    "T_Agarrado";
      NOP   0;
      NOP   0;
      NOP   0;
      NOP   0;
      A     L 18.0;
      AN    "40Y4";
      AN    "40Y5";
      AN    "40Y6";
      L     S5T#1S;
      SD    "T_Soltado";
      NOP   0;
      NOP   0;
      NOP   0;
      NOP   0;
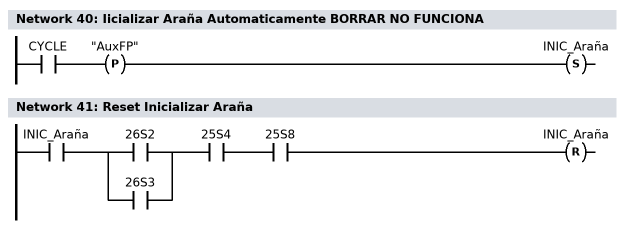
NETWORK
TITLE = Iicializar Araña Automaticamente BORRAR NO FUNCIONA
      A     "CYCLE";
      FP    "AuxFP";
      S     "INIC_Araña";
NETWORK
TITLE = Reset Inicializar Araña
      A     "INIC_Araña";
      A(;
      O     "26S2";
      O     "26S3";
      );
      A     "25S4";
      A     "25S8";
      R     "INIC_Araña";
END_FUNCTION

FUNCTION "Descarga" : VOID	// FC 40
//LUC - 13/08/2020
VERSION : 0.1
VAR_TEMP
  SECU : BOOL ;	//Sécurité mécanique du mouvement
  AUX_SECU : BOOL ;
  NMVT : INT ;	//Numero Mouvement
  M01 : BOOL ;
  FEN_P : DINT ;
  FEN_N : DINT ;
END_VAR
BEGIN
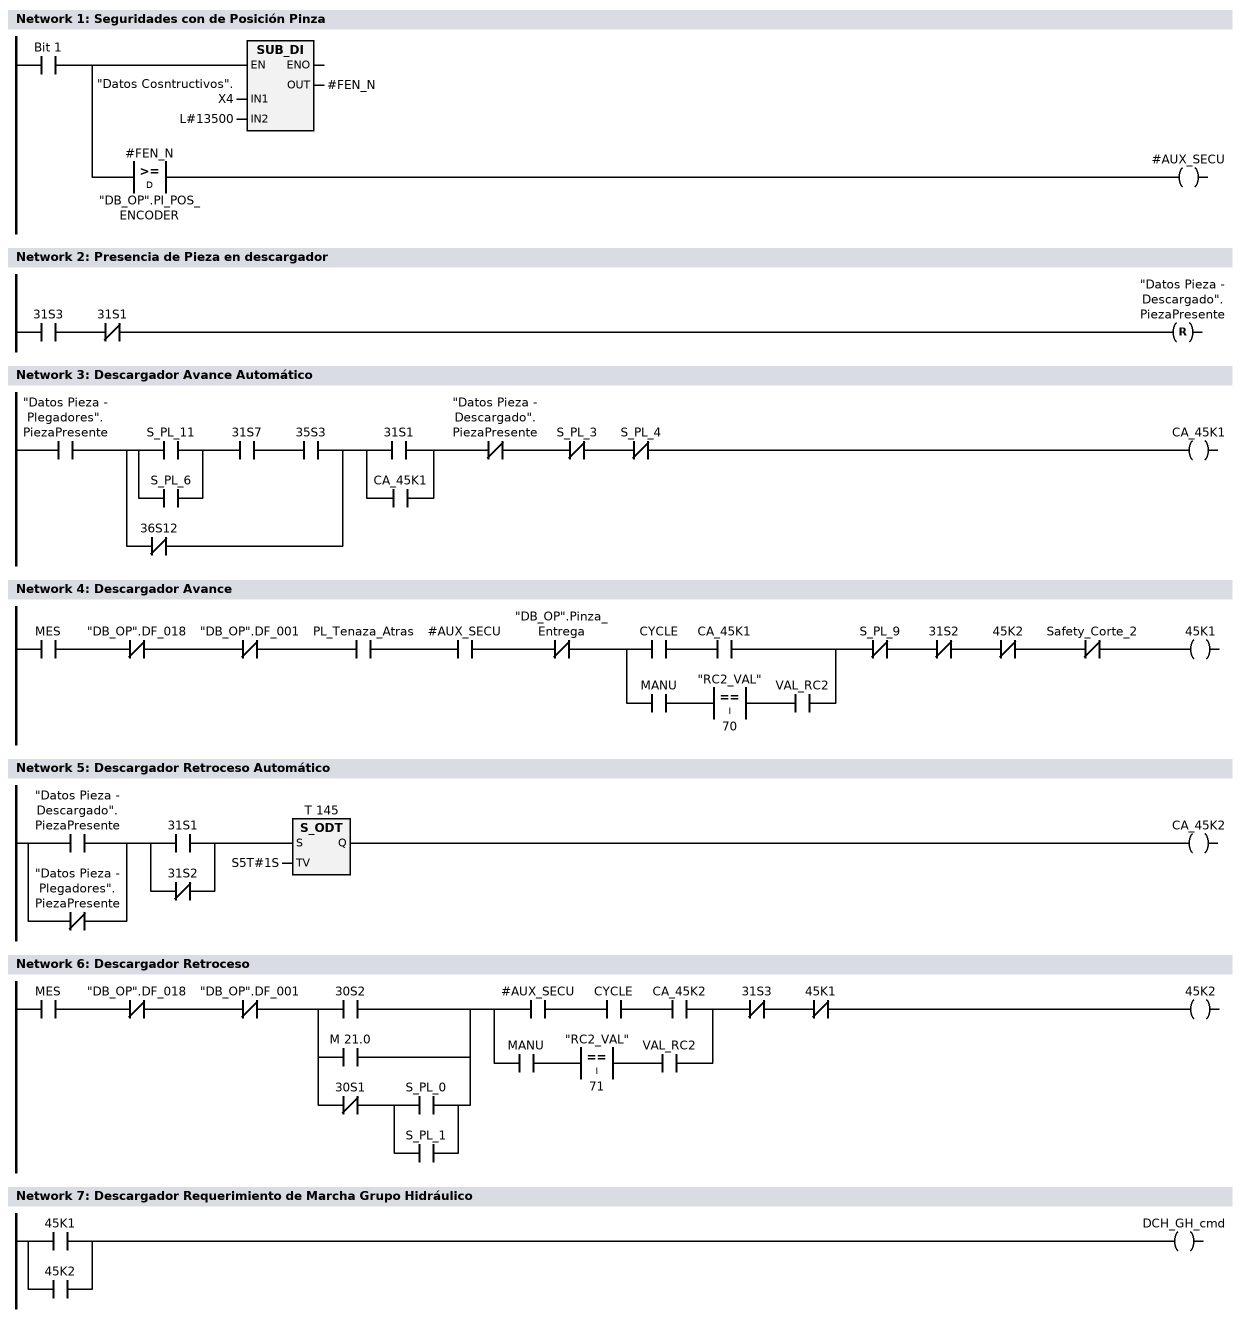
NETWORK
TITLE = Seguridades con de Posición Pinza
      A     "Bit 1";
      =     L 14.0;
      A     L 14.0;
      JNB   _001;
      L     "Datos Cosntructivos".X4;
      L     L#13500;
      -D;
      T     #FEN_N;
_001: NOP   0;
      A     L 14.0;
      A(;
      L     #FEN_N;
      L     "DB_OP".PI_POS_ENCODER;
      >=D;
      );
      =     #AUX_SECU;
NETWORK
TITLE = Presencia de Pieza en descargador
      A     "31S3";
      AN    "31S1";
      R     "Datos Pieza - Descargado".PiezaPresente;
NETWORK
TITLE = Descargador Avance Automático
      A     "Datos Pieza - Plegadores".PiezaPresente;
      A(;
      A(;
      O     "S_PL_11";
      O     "S_PL_6";
      );
      A     "31S7";
      A     "35S3";
      ON    "36S12";
      );
      A(;
      O     "31S1";
      O     "CA_45K1";
      );
      AN    "Datos Pieza - Descargado".PiezaPresente;
      AN    "S_PL_3";
      AN    "S_PL_4";
      =     "CA_45K1";
NETWORK
TITLE = Descargador Avance
      A     "MES";
      AN    "DB_OP".DF_018;
      AN    "DB_OP".DF_001;
      A     "PL_Tenaza_Atras";
      A     #AUX_SECU;
      AN    "DB_OP".Pinza_Entrega;
      A(;
      A     "CYCLE";
      A     "CA_45K1";
      O;
      A     "MANU";
      A(;
      L     "RC2_VAL";
      L     70;
      ==I;
      );
      A     "VAL_RC2";
      );
      AN    "S_PL_9";
      AN    "31S2";
      AN    "45K2";
      AN    "Safety_Corte_2";
      =     "45K1";
NETWORK
TITLE = Descargador Retroceso Automático
      A(;
      O     "Datos Pieza - Descargado".PiezaPresente;
      ON    "Datos Pieza - Plegadores".PiezaPresente;
      );
      A(;
      O     "31S1";
      ON    "31S2";
      );
      L     S5T#1S;
      SD    T 145;
      NOP   0;
      NOP   0;
      NOP   0;
      A     T 145;
      =     "CA_45K2";
NETWORK
TITLE = Descargador Retroceso
      A     "MES";
      AN    "DB_OP".DF_018;
      AN    "DB_OP".DF_001;
      A(;
      O     "30S2";
      O     M 21.0;
      O;
      AN    "30S1";
      A(;
      O     "S_PL_0";
      O     "S_PL_1";
      );
      );
      A(;
      A     #AUX_SECU;
      A     "CYCLE";
      A     "CA_45K2";
      O;
      A     "MANU";
      A(;
      L     "RC2_VAL";
      L     71;
      ==I;
      );
      A     "VAL_RC2";
      );
      AN    "31S3";
      AN    "45K1";
      =     "45K2";
NETWORK
TITLE = Descargador Requerimiento de Marcha Grupo Hidráulico
      O     "45K1";
      O     "45K2";
      =     "DCH_GH_cmd";
END_FUNCTION

FUNCTION "Gestión de Datos" : VOID	// FC 51
VERSION : 0.1
VAR_TEMP
  Aux_Bucle : INT ;
END_VAR
BEGIN
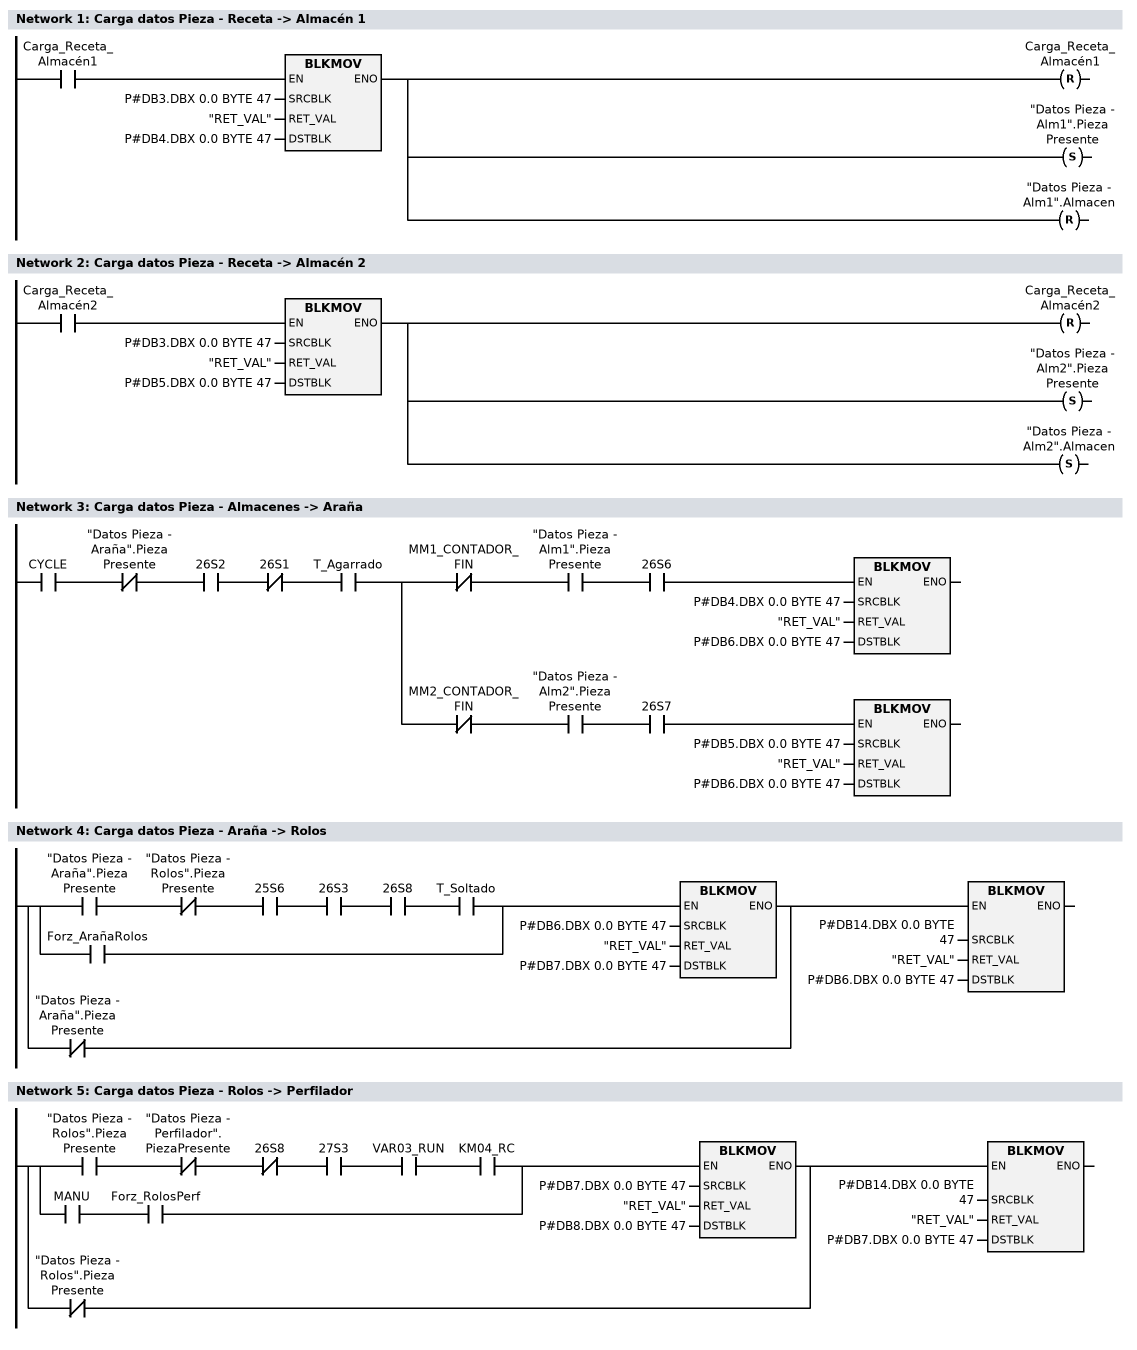
NETWORK
TITLE = Carga datos Pieza - Receta -> Almacén 1
      A     "Carga_Receta_Almacén1";
      JNB   _001;
      CALL  "BLKMOV" (
           SRCBLK                   := P#DB3.DBX 0.0 BYTE 47,
           RET_VAL                  := "RET_VAL",
           DSTBLK                   := P#DB4.DBX 0.0 BYTE 47);
_001: A     BR;
      R     "Carga_Receta_Almacén1";
      S     "Datos Pieza - Alm1".PiezaPresente;
      R     "Datos Pieza - Alm1".Almacen;
NETWORK
TITLE = Carga datos Pieza - Receta -> Almacén 2
      A     "Carga_Receta_Almacén2";
      JNB   _002;
      CALL  "BLKMOV" (
           SRCBLK                   := P#DB3.DBX 0.0 BYTE 47,
           RET_VAL                  := "RET_VAL",
           DSTBLK                   := P#DB5.DBX 0.0 BYTE 47);
_002: A     BR;
      R     "Carga_Receta_Almacén2";
      S     "Datos Pieza - Alm2".PiezaPresente;
      S     "Datos Pieza - Alm2".Almacen;
NETWORK
TITLE = Carga datos Pieza - Almacenes -> Araña
      A     "CYCLE";
      AN    "Datos Pieza - Araña".PiezaPresente;
      A     "26S2";
      AN    "26S1";
      A     "T_Agarrado";
      =     L 2.0;
      A     L 2.0;
      AN    "MM1_CONTADOR_FIN";
      A     "Datos Pieza - Alm1".PiezaPresente;
      A     "26S6";
      JNB   _003;
      CALL  "BLKMOV" (
           SRCBLK                   := P#DB4.DBX 0.0 BYTE 47,
           RET_VAL                  := "RET_VAL",
           DSTBLK                   := P#DB6.DBX 0.0 BYTE 47);
_003: NOP   0;
      A     L 2.0;
      AN    "MM2_CONTADOR_FIN";
      A     "Datos Pieza - Alm2".PiezaPresente;
      A     "26S7";
      JNB   _004;
      CALL  "BLKMOV" (
           SRCBLK                   := P#DB5.DBX 0.0 BYTE 47,
           RET_VAL                  := "RET_VAL",
           DSTBLK                   := P#DB6.DBX 0.0 BYTE 47);
_004: NOP   0;
NETWORK
TITLE = Carga datos Pieza - Araña -> Rolos
      A(;
      O(;
      A(;
      A     "Datos Pieza - Araña".PiezaPresente;
      AN    "Datos Pieza - Rolos".PiezaPresente;
      A     "25S6";
      A     "26S3";
      A     "26S8";
      A     "T_Soltado";
      O     "Forz_ArañaRolos";
      );
      JNB   _005;
      CALL  "BLKMOV" (
           SRCBLK                   := P#DB6.DBX 0.0 BYTE 47,
           RET_VAL                  := "RET_VAL",
           DSTBLK                   := P#DB7.DBX 0.0 BYTE 47);
_005: A     BR;
      );
      ON    "Datos Pieza - Araña".PiezaPresente;
      );
      JNB   _006;
      CALL  "BLKMOV" (
           SRCBLK                   := P#DB14.DBX 0.0 BYTE 47,
           RET_VAL                  := "RET_VAL",
           DSTBLK                   := P#DB6.DBX 0.0 BYTE 47);
_006: NOP   0;
NETWORK
TITLE = Carga datos Pieza - Rolos -> Perfilador
      A(;
      O(;
      A(;
      A     "Datos Pieza - Rolos".PiezaPresente;
      AN    "Datos Pieza - Perfilador".PiezaPresente;
      AN    "26S8";
      A     "27S3";
      A     "VAR03_RUN";
      A     "KM04_RC";
      O;
      A     "MANU";
      A     "Forz_RolosPerf";
      );
      JNB   _007;
      CALL  "BLKMOV" (
           SRCBLK                   := P#DB7.DBX 0.0 BYTE 47,
           RET_VAL                  := "RET_VAL",
           DSTBLK                   := P#DB8.DBX 0.0 BYTE 47);
_007: A     BR;
      );
      ON    "Datos Pieza - Rolos".PiezaPresente;
      );
      JNB   _008;
      CALL  "BLKMOV" (
           SRCBLK                   := P#DB14.DBX 0.0 BYTE 47,
           RET_VAL                  := "RET_VAL",
           DSTBLK                   := P#DB7.DBX 0.0 BYTE 47);
_008: NOP   0;
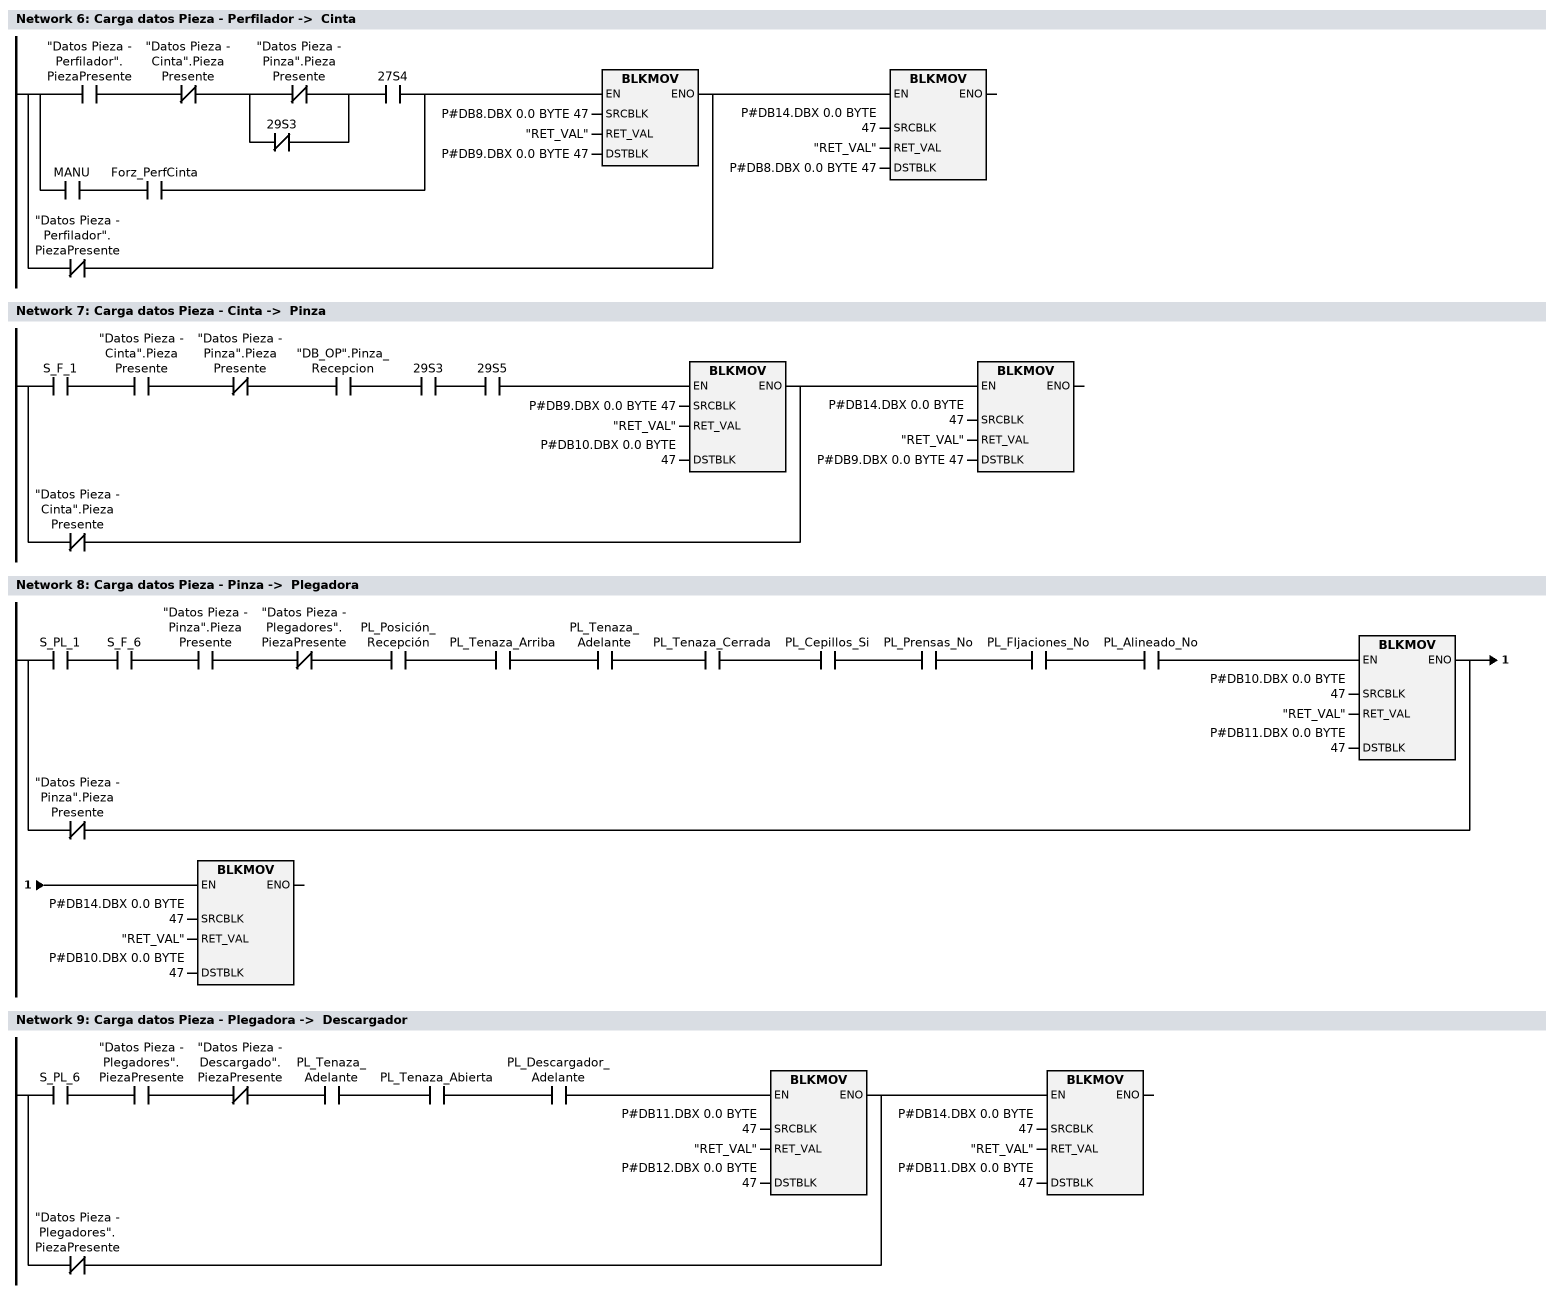
NETWORK
TITLE = Carga datos Pieza - Perfilador ->  Cinta
      A(;
      O(;
      A(;
      A     "Datos Pieza - Perfilador".PiezaPresente;
      AN    "Datos Pieza - Cinta".PiezaPresente;
      A(;
      ON    "Datos Pieza - Pinza".PiezaPresente;
      ON    "29S3";
      );
      A     "27S4";
      O;
      A     "MANU";
      A     "Forz_PerfCinta";
      );
      JNB   _009;
      CALL  "BLKMOV" (
           SRCBLK                   := P#DB8.DBX 0.0 BYTE 47,
           RET_VAL                  := "RET_VAL",
           DSTBLK                   := P#DB9.DBX 0.0 BYTE 47);
_009: A     BR;
      );
      ON    "Datos Pieza - Perfilador".PiezaPresente;
      );
      JNB   _00a;
      CALL  "BLKMOV" (
           SRCBLK                   := P#DB14.DBX 0.0 BYTE 47,
           RET_VAL                  := "RET_VAL",
           DSTBLK                   := P#DB8.DBX 0.0 BYTE 47);
_00a: NOP   0;
NETWORK
TITLE = Carga datos Pieza - Cinta ->  Pinza
      A(;
      O(;
      A     "S_F_1";
      A     "Datos Pieza - Cinta".PiezaPresente;
      AN    "Datos Pieza - Pinza".PiezaPresente;
      A     "DB_OP".Pinza_Recepcion;
      A     "29S3";
      A     "29S5";
      JNB   _00b;
      CALL  "BLKMOV" (
           SRCBLK                   := P#DB9.DBX 0.0 BYTE 47,
           RET_VAL                  := "RET_VAL",
           DSTBLK                   := P#DB10.DBX 0.0 BYTE 47);
_00b: A     BR;
      );
      ON    "Datos Pieza - Cinta".PiezaPresente;
      );
      JNB   _00c;
      CALL  "BLKMOV" (
           SRCBLK                   := P#DB14.DBX 0.0 BYTE 47,
           RET_VAL                  := "RET_VAL",
           DSTBLK                   := P#DB9.DBX 0.0 BYTE 47);
_00c: NOP   0;
NETWORK
TITLE = Carga datos Pieza - Pinza ->  Plegadora
      A(;
      O(;
      A     "S_PL_1";
      A     "S_F_6";
      A     "Datos Pieza - Pinza".PiezaPresente;
      AN    "Datos Pieza - Plegadores".PiezaPresente;
      A     "PL_Posición_Recepción";
      A     "PL_Tenaza_Arriba";
      A     "PL_Tenaza_Adelante";
      A     "PL_Tenaza_Cerrada";
      A     "PL_Cepillos_Si";
      A     "PL_Prensas_No";
      A     "PL_FIjaciones_No";
      A     "PL_Alineado_No";
      JNB   _00d;
      CALL  "BLKMOV" (
           SRCBLK                   := P#DB10.DBX 0.0 BYTE 47,
           RET_VAL                  := "RET_VAL",
           DSTBLK                   := P#DB11.DBX 0.0 BYTE 47);
_00d: A     BR;
      );
      ON    "Datos Pieza - Pinza".PiezaPresente;
      );
      JNB   _00e;
      CALL  "BLKMOV" (
           SRCBLK                   := P#DB14.DBX 0.0 BYTE 47,
           RET_VAL                  := "RET_VAL",
           DSTBLK                   := P#DB10.DBX 0.0 BYTE 47);
_00e: NOP   0;
NETWORK
TITLE = Carga datos Pieza - Plegadora ->  Descargador
      A(;
      O(;
      A     "S_PL_6";
      A     "Datos Pieza - Plegadores".PiezaPresente;
      AN    "Datos Pieza - Descargado".PiezaPresente;
      A     "PL_Tenaza_Adelante";
      A     "PL_Tenaza_Abierta";
      A     "PL_Descargador_Adelante";
      JNB   _00f;
      CALL  "BLKMOV" (
           SRCBLK                   := P#DB11.DBX 0.0 BYTE 47,
           RET_VAL                  := "RET_VAL",
           DSTBLK                   := P#DB12.DBX 0.0 BYTE 47);
_00f: A     BR;
      );
      ON    "Datos Pieza - Plegadores".PiezaPresente;
      );
      JNB   _010;
      CALL  "BLKMOV" (
           SRCBLK                   := P#DB14.DBX 0.0 BYTE 47,
           RET_VAL                  := "RET_VAL",
           DSTBLK                   := P#DB11.DBX 0.0 BYTE 47);
_010: NOP   0;
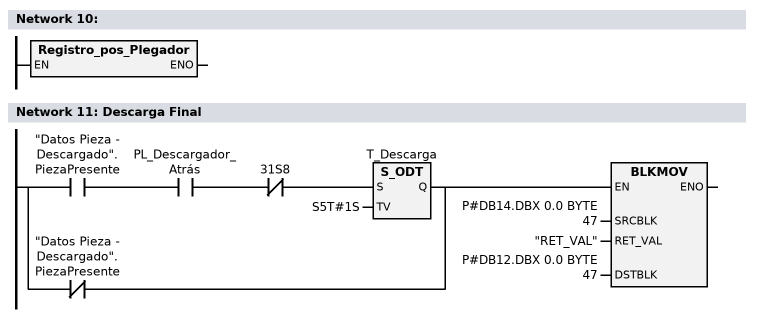
NETWORK
TITLE =
      CALL  "Registro_pos_Plegador";
      NOP   0;
NETWORK
TITLE = Descarga Final
      A(;
      O(;
      A     "Datos Pieza - Descargado".PiezaPresente;
      A     "PL_Descargador_Atrás";
      AN    "31S8";
      L     S5T#1S;
      SD    "T_Descarga";
      NOP   0;
      NOP   0;
      NOP   0;
      A     "T_Descarga";
      );
      ON    "Datos Pieza - Descargado".PiezaPresente;
      );
      JNB   _011;
      CALL  "BLKMOV" (
           SRCBLK                   := P#DB14.DBX 0.0 BYTE 47,
           RET_VAL                  := "RET_VAL",
           DSTBLK                   := P#DB12.DBX 0.0 BYTE 47);
_011: NOP   0;
END_FUNCTION

// FC 150: know-how protected block, not included

DATA_BLOCK "Tendencia"	// DB 1
VERSION : 0.1
  STRUCT
   T_H1 : REAL ;	//Tiempo Heladera 1
   T_H2 : REAL ;	//Tiempo Heladera 2
   T_H3 : REAL ;	//Tiempo Heladera 3
   T_H4 : REAL ;	//Tiempo Heladera 4
   T_H5 : REAL ;	//Tiempo Heladera 5
   T_H6 : REAL ;	//Tiempo Heladera 6
   T_H7 : REAL ;	//Tiempo Heladera 7
   T_H8 : REAL ;	//Tiempo Heladera 8
   T_H9 : REAL ;	//Tiempo Heladera 9
   T_H10 : REAL ;	//Tiempo Heladera 10
   T_PROM : REAL ;	//Tiempo Promedio
   CANT_PROV : REAL ;	//Cantidad Provisoria
   HELxHORAINST : REAL ;	//Heladeras por hora (Instantáneo)
   TiempoServosPL : REAL ;	//Tiempo Demorado por Servos Plegadora
   TiempoHidrPL : REAL ;	//Tiempo Demorado por movimientos hidráulicos Plegadora
   TiempoAirePL : REAL ;	//Tiempo Demorado por movimmientos neumáticos
   TiempoDescargador : REAL ;	//Tiempo Demorado por descargador
   TiempoServosPL1_PARCIAL : REAL ;	//Tiempo Demorado por Servos Plegadora Parcial
   TiempoHidrPL1_PARCIAL : REAL ;	//Tiempo Demorado por movimientos hidráulicos Plegadora Parcial
   TiempoAirePL1_PARCIAL : REAL ;	//Tiempo Demorado por movimmientos neumáticos Parcial
   TiempoDescargad_PARCIAL : REAL ;	//Tiempo Demorado por descargador Parcial
  END_STRUCT ;	
BEGIN
END_DATA_BLOCK

DATA_BLOCK "EncóderPerfilador"	// DB 2
VERSION : 0.1
  STRUCT
   Medicion_Operador_Perf : REAL  := 6.670000e+002;	//Medición tomada por operador en perfiladores
   Aux_Medicion : REAL ;
   Deshabilitar : BOOL ;
   AuX_EMR : REAL ;
  END_STRUCT ;	
BEGIN
END_DATA_BLOCK

DATA_BLOCK "Datos Pieza - Receta"	// DB 3
AUTHOR : EMR
NAME : eProC
VERSION : 0.1
  STRUCT
   A : INT ;
   B : INT ;
   C : INT ;
   D : INT ;
   F1 : INT ;
   F2 : INT ;
   F3 : INT ;
   F4 : INT ;
   PL1_1 : INT ;
   PL1_2 : INT ;
   PL2_1 : INT ;
   PL2_2 : INT ;
   NOMBRE : STRING  [20 ];
   PiezaPresente : BOOL ;
   Almacen : BOOL ;	//0=almacen 1 / 1=almacen 2
  END_STRUCT ;	
BEGIN
END_DATA_BLOCK

DATA_BLOCK "Datos Pieza - Alm1"	// DB 4
AUTHOR : EMR
NAME : eProC
VERSION : 0.1
  STRUCT
   A : INT ;
   B : INT ;
   C : INT ;
   D : INT ;
   F1 : INT ;
   F2 : INT ;
   F3 : INT ;
   F4 : INT ;
   PL1_1 : INT ;
   PL1_2 : INT ;
   PL2_1 : INT ;
   PL2_2 : INT ;
   NOMBRE : STRING  [20 ];
   PiezaPresente : BOOL ;
   Almacen : BOOL ;	//0=almacen 1 / 1=almacen 2
  END_STRUCT ;	
BEGIN
END_DATA_BLOCK

DATA_BLOCK "Datos Pieza - Alm2"	// DB 5
AUTHOR : EMR
NAME : eProC
VERSION : 0.1
  STRUCT
   A : INT ;
   B : INT ;
   C : INT ;
   D : INT ;
   F1 : INT ;
   F2 : INT ;
   F3 : INT ;
   F4 : INT ;
   PL1_1 : INT ;
   PL1_2 : INT ;
   PL2_1 : INT ;
   PL2_2 : INT ;
   NOMBRE : STRING  [20 ];
   PiezaPresente : BOOL ;
   Almacen : BOOL  := TRUE;	//0=almacen 1 / 1=almacen 2
  END_STRUCT ;	
BEGIN
END_DATA_BLOCK

DATA_BLOCK "Datos Pieza - Araña"	// DB 6
AUTHOR : EMR
NAME : eProC
VERSION : 0.1
  STRUCT
   A : INT ;
   B : INT ;
   C : INT ;
   D : INT ;
   F1 : INT ;
   F2 : INT ;
   F3 : INT ;
   F4 : INT ;
   PL1_1 : INT ;
   PL1_2 : INT ;
   PL2_1 : INT ;
   PL2_2 : INT ;
   NOMBRE : STRING  [20 ];
   PiezaPresente : BOOL ;
   Almacen : BOOL ;	//0=almacen 1 / 1=almacen 2
  END_STRUCT ;	
BEGIN
END_DATA_BLOCK

DATA_BLOCK "Datos Pieza - Rolos"	// DB 7
AUTHOR : EMR
NAME : eProC
VERSION : 0.1
  STRUCT
   A : INT ;
   B : INT ;
   C : INT ;
   D : INT ;
   F1 : INT ;
   F2 : INT ;
   F3 : INT ;
   F4 : INT ;
   PL1_1 : INT ;
   PL1_2 : INT ;
   PL2_1 : INT ;
   PL2_2 : INT ;
   NOMBRE : STRING  [20 ];
   PiezaPresente : BOOL ;
   Almacen : BOOL ;	//0=almacen 1 / 1=almacen 2
  END_STRUCT ;	
BEGIN
END_DATA_BLOCK

DATA_BLOCK "Datos Pieza - Perfilador"	// DB 8
AUTHOR : EMR
NAME : eProC
VERSION : 0.1
  STRUCT
   A : INT ;
   B : INT ;
   C : INT ;
   D : INT ;
   F1 : INT ;
   F2 : INT ;
   F3 : INT ;
   F4 : INT ;
   PL1_1 : INT ;
   PL1_2 : INT ;
   PL2_1 : INT ;
   PL2_2 : INT ;
   NOMBRE : STRING  [20 ];
   PiezaPresente : BOOL ;
   Almacen : BOOL ;	//0=almacen 1 / 1=almacen 2
  END_STRUCT ;	
BEGIN
END_DATA_BLOCK

DATA_BLOCK "Datos Pieza - Cinta"	// DB 9
AUTHOR : EMR
NAME : eProC
VERSION : 0.1
  STRUCT
   A : INT ;
   B : INT ;
   C : INT ;
   D : INT ;
   F1 : INT ;
   F2 : INT ;
   F3 : INT ;
   F4 : INT ;
   PL1_1 : INT ;
   PL1_2 : INT ;
   PL2_1 : INT ;
   PL2_2 : INT ;
   NOMBRE : STRING  [20 ];
   PiezaPresente : BOOL ;
   Almacen : BOOL ;	//0=almacen 1 / 1=almacen 2
  END_STRUCT ;	
BEGIN
END_DATA_BLOCK

DATA_BLOCK "Datos Pieza - Pinza"	// DB 10
AUTHOR : EMR
NAME : eProC
VERSION : 0.1
  STRUCT
   A : INT ;
   B : INT ;
   C : INT ;
   D : INT ;
   F1 : INT ;
   F2 : INT ;
   F3 : INT ;
   F4 : INT ;
   PL1_1 : INT ;
   PL1_2 : INT ;
   PL2_1 : INT ;
   PL2_2 : INT ;
   NOMBRE : STRING  [20 ];
   PiezaPresente : BOOL ;
   Almacen : BOOL ;	//0=almacen 1 / 1=almacen 2
  END_STRUCT ;	
BEGIN
END_DATA_BLOCK

DATA_BLOCK "Datos Pieza - Plegadores"	// DB 11
AUTHOR : EMR
NAME : eProC
VERSION : 0.1
  STRUCT
   A : INT ;
   B : INT ;
   C : INT ;
   D : INT ;
   F1 : INT ;
   F2 : INT ;
   F3 : INT ;
   F4 : INT ;
   PL1_1 : INT ;
   PL1_2 : INT ;
   PL2_1 : INT ;
   PL2_2 : INT ;
   NOMBRE : STRING  [20 ];
   PiezaPresente : BOOL ;
   Almacen : BOOL ;	//0=almacen 1 / 1=almacen 2
  END_STRUCT ;	
BEGIN
END_DATA_BLOCK

DATA_BLOCK "Datos Pieza - Descargado"	// DB 12
AUTHOR : EMR
NAME : eProC
VERSION : 0.1
  STRUCT
   A : INT ;
   B : INT ;
   C : INT ;
   D : INT ;
   F1 : INT ;
   F2 : INT ;
   F3 : INT ;
   F4 : INT ;
   PL1_1 : INT ;
   PL1_2 : INT ;
   PL2_1 : INT ;
   PL2_2 : INT ;
   NOMBRE : STRING  [20 ];
   PiezaPresente : BOOL ;
   Almacen : BOOL ;	//0=almacen 1 / 1=almacen 2
  END_STRUCT ;	
BEGIN
END_DATA_BLOCK

DATA_BLOCK "Posiciones_Pinza"	// DB 13
VERSION : 0.1
  STRUCT
   Pos_Recepcion : DINT ;
   Pos_E1H1 : DINT ;
   Pos_E1H2 : DINT ;
   Pos_E2H1 : DINT ;
   Pos_E2H2 : DINT ;
   Pos_Entrega : DINT ;
  END_STRUCT ;	
BEGIN
END_DATA_BLOCK

DATA_BLOCK "Datos Pieza - VACIO"	// DB 14
VERSION : 0.1
  STRUCT
   A : INT ;
   B : INT ;
   C : INT ;
   D : INT ;
   F1 : INT ;
   F2 : INT ;
   F3 : INT ;
   F4 : INT ;
   PL1_1 : INT ;
   PL1_2 : INT ;
   PL2_1 : INT ;
   PL2_2 : INT ;
   NOMBRE : STRING  [20 ];
   PiezaPresente : BOOL ;
  END_STRUCT ;	
BEGIN
END_DATA_BLOCK

DATA_BLOCK "Ultimo Estado"	// DB 15
VERSION : 0.1
  STRUCT
   Plegadora : WORD ;
   Formador : WORD ;
   Pinza : WORD ;
  END_STRUCT ;	
BEGIN
END_DATA_BLOCK

DATA_BLOCK "Datos Cosntructivos"	// DB 16
VERSION : 0.1
  STRUCT
   X1 : DINT  := L#21300;	//Distancia entre Herramientas Formador
   X2 : DINT  := L#77100;	//Distancia entre H1 y Cero de Pinza
   X3 : DINT  := L#297200;	//Distancia entre Cero de Pinza y Tenaza plegadora
   X4 : DINT  := L#200000;	//Distancia entre Cero de Pinza y Descargador
   X5 : DINT  := L#520000;	//Distancia entre Cero de Pinza y Máximo Recorrido Pinza
   X6 : DINT  := L#250000;	//Distancia entre Tenaza Plegadora y Máximo Recorrido de Plegador
   X7 : DINT  := L#45536;	//Distancia entre Tenaza Plegadora y Mínimo Recorrido de Plegador
   X8 : DINT  := L#55500;	//Distancia entre Prensa Plegadores y Alineadores
  END_STRUCT ;	
BEGIN
   X1 := L#21300;
   X2 := L#77100;
   X3 := L#297200;
   X4 := L#200000;
   X5 := L#520000;
   X6 := L#250000;
   X7 := L#45536;
   X8 := L#55500;
END_DATA_BLOCK

DATA_BLOCK "Posiciones Pinza 00"	// DB 17
VERSION : 0.1
  STRUCT
   Pos_Recepcion : DINT ;
   Pos_E1H1 : DINT  := L#1000;
   Pos_E1H2 : DINT  := L#1000;
   Pos_E2H1 : DINT  := L#1000;
   Pos_E2H2 : DINT  := L#1000;
   Pos_Entrega : DINT  := L#1000;
  END_STRUCT ;	
BEGIN
   Pos_E1H1 := L#1000;
   Pos_E1H2 := L#1000;
   Pos_E2H1 := L#1000;
   Pos_E2H2 := L#1000;
   Pos_Entrega := L#1000;
END_DATA_BLOCK

DATA_BLOCK "Posiciones_Pinza_Ant"	// DB 18
VERSION : 0.1
  STRUCT
   Pos_Recepcion : DINT ;
   Pos_E1H1 : DINT ;
   Pos_E1H2 : DINT ;
   Pos_E2H1 : DINT ;
   Pos_E2H2 : DINT ;
   Pos_Entrega : DINT ;
  END_STRUCT ;	
BEGIN
END_DATA_BLOCK

DATA_BLOCK "DB Asistencia"	// DB 19
VERSION : 0.1
  STRUCT
   IncF_A1 : INT ;	//Operador Solicita Incremento de F Almacén 1
   DecF_A1 : INT ;	//Operador Solicita Decremento de F Almacén 1
   IncF_A2 : INT ;	//Operador Solicita Incremento de F Almacén 2
   DecF_A2 : INT ;	//Operador Solicita Decremento de F Almacén 2
   ResolucF : INT ;	//Resolución Incremento/Decremento F
   IncPL_A1 : INT ;	//Operador Solicita Incremento de PL Almacén 1
   DecPL_A1 : INT ;	//Operador Solicita Decremento de PL Almacén 1
   IncPL_A2 : INT ;	//Operador Solicita Incremento de PL Almacén 2
   DecPL_A2 : INT ;	//Operador Solicita Decremento de PL Almacén 2
   ResolucPL : INT ;	//Resolución Incremento/Decremento PL
  END_STRUCT ;	
BEGIN
END_DATA_BLOCK

DATA_BLOCK "ReglasBalluff"	// DB 20
AUTHOR : FRD
VERSION : 0.1
  STRUCT
   PL1_COD_COEF : DINT  := L#1;	//Multiplicador para obtener posición Plegador 1 con regla Balluff
   PL1_POS_CONSIGNA_INICIO : DINT ;	//Offset para obtener posición Plegador 1 con regla Balluff
   PL2_COD_COEF : DINT  := L#1;	//Multiplicador para obtener posición Plegador 2 con regla Balluff
   PL2_POS_CONSIGNA_INICIO : DINT ;	//Offset para obtener posición Plegador 2 con regla Balluff
   PI_COD_COEF : DINT  := L#1;	//Multiplicador para obtener posición Pinza con regla Balluff
   PI_POS_CONSIGNA_INICIO : DINT ;	//Offset para obtener posición Pinza con regla Balluff
   Reglas_ON : BOOL ;	//1: Habilita el uso de las reglas. 0: Habilita uso de Encoders
  END_STRUCT ;	
BEGIN
   PL1_COD_COEF := L#1;
   PL2_COD_COEF := L#1;
   PI_COD_COEF := L#1;
END_DATA_BLOCK

DATA_BLOCK "Referenciado"	// DB 21
VERSION : 0.1
  STRUCT
   Homing_PL1 : BOOL ;	//Secuencia referenciado PL1 en proceso
   Homing_PL2 : BOOL ;	//Secuencia referenciado PL1 en proceso
   HMI_SolRef_PL1 : BOOL ;	//Solicitud referenciado PL1 (desde panel)
   HMI_SolRef_PL2 : BOOL ;	//Solicitud referenciado PL2 (desde panel)
   Reserva4 : BOOL ;
   Reserva5 : BOOL ;
   Reserva6 : BOOL ;
   Reserva7 : BOOL ;
  END_STRUCT ;	
BEGIN
END_DATA_BLOCK

DATA_BLOCK "Posiciones_Pinza_Ant2"	// DB 23
NAME : eProC
VERSION : 0.1
  STRUCT
   Pos_Recepcion : DINT ;
   Pos_E1H1 : DINT ;
   Pos_E1H2 : DINT ;
   Pos_E2H1 : DINT ;
   Pos_E2H2 : DINT ;
   Pos_Entrega : DINT ;
  END_STRUCT ;	
BEGIN
END_DATA_BLOCK

DATA_BLOCK "Posiciones_Pinza_Ant3"	// DB 24
NAME : eProC
VERSION : 0.1
  STRUCT
   Pos_Recepcion : DINT ;
   Pos_E1H1 : DINT ;
   Pos_E1H2 : DINT ;
   Pos_E2H1 : DINT ;
   Pos_E2H2 : DINT ;
   Pos_Entrega : DINT ;
  END_STRUCT ;	
BEGIN
END_DATA_BLOCK

DATA_BLOCK "PosReal_Pinza"	// DB 25
NAME : eProC
VERSION : 0.1
  STRUCT
   Pos_Recepcion : DINT ;
   Pos_E1H1 : DINT ;
   Pos_E1H2 : DINT ;
   Pos_E2H1 : DINT ;
   Pos_E2H2 : DINT ;
   Pos_Entrega : DINT ;
  END_STRUCT ;	
BEGIN
END_DATA_BLOCK

DATA_BLOCK "PosReal_Pinza_Ant"	// DB 26
NAME : eProC
VERSION : 0.1
  STRUCT
   Pos_Recepcion : DINT ;
   Pos_E1H1 : DINT ;
   Pos_E1H2 : DINT ;
   Pos_E2H1 : DINT ;
   Pos_E2H2 : DINT ;
   Pos_Entrega : DINT ;
  END_STRUCT ;	
BEGIN
END_DATA_BLOCK

DATA_BLOCK "PosReal_Pinza_Ant2"	// DB 27
NAME : eProC
VERSION : 0.1
  STRUCT
   Pos_Recepcion : DINT ;
   Pos_E1H1 : DINT ;
   Pos_E1H2 : DINT ;
   Pos_E2H1 : DINT ;
   Pos_E2H2 : DINT ;
   Pos_Entrega : DINT ;
  END_STRUCT ;	
BEGIN
END_DATA_BLOCK

DATA_BLOCK "PosReal_Pinza_Ant3"	// DB 28
NAME : eProC
VERSION : 0.1
  STRUCT
   Pos_Recepcion : DINT ;
   Pos_E1H1 : DINT ;
   Pos_E1H2 : DINT ;
   Pos_E2H1 : DINT ;
   Pos_E2H2 : DINT ;
   Pos_Entrega : DINT ;
  END_STRUCT ;	
BEGIN
END_DATA_BLOCK

DATA_BLOCK "Error_Pinza_Ant"	// DB 29
NAME : eProC
VERSION : 0.1
  STRUCT
   Pos_Recepcion : DINT ;
   Pos_E1H1 : DINT ;
   Pos_E1H2 : DINT ;
   Pos_E2H1 : DINT ;
   Pos_E2H2 : DINT ;
   Pos_Entrega : DINT ;
  END_STRUCT ;	
BEGIN
END_DATA_BLOCK

DATA_BLOCK "DB_OP"	// DB 50
VERSION : 0.1
  STRUCT
   P_DEFAUT : BOOL ;
   ACQ_DEFAUT : BOOL ;
   OP_SELMANU1 : BOOL ;
   OP_SELMANU2 : BOOL ;
   MODE : INT ;	//Modo de Marcha
   RC1 : INT ;
   RC2 : INT ;
   DB_VAR : ARRAY  [1 .. 21 ] OF //Variables temporales
   INT  := 0;
   DF_001 : BOOL ;	//Falla térmica en motor refrigeración de grupo hidráulico Plegado
   DF_002 : BOOL ;	//Falla Almacenes Deshabilitados
   DF_003 : BOOL ;	//Falla Alimentación Motor Intercambio de Almacenes
   DF_004 : BOOL ;	//Falla en Variador Transporte de Araña
   DF_005 : BOOL ;	//Falla en Variador Transporte Rolos
   DF_006 : BOOL ;	//Falla en Control Unit Perfiladores
   DF_007 : BOOL ;	//Falla en etapa de Potencia de variadores Perfiladores
   DF_008 : BOOL ;	//CU Plegadora - Falla Presente
   DF_009 : BOOL ;	//CU Plegadora - Falla Safety Presente
   DF_010 : BOOL ;	//Falla térmica en bomba de lubricación de Perfiladores
   DF_011 : BOOL ;	//Falla térmica en grupo hidraulico de freno Perfiladores
   DF_012 : BOOL ;	//Falla térmica en motor Ajuste de ancho de Perfiladores
   DF_013 : BOOL ;	//Falla en Variador Transporte Cinta
   DF_014 : BOOL ;	//Falla térmica en motor ajuste de ancho en etapa de formado
   DF_015 : BOOL ;	//Falla Rectificador de variadores Plegadores
   DF_016 : BOOL ;	//Falla límite de Seguridad en Plegador 1
   DF_017 : BOOL ;	//Falla límite de Seguridad en Plegador 2
   DF_018 : BOOL ;	//Falla térmica en motor grupo hidráulico Plegadora
   DF_019 : BOOL ;	//Falla térmica en freno de motor ajuste de ancho en etapa de Form
   DF_020 : BOOL ;	//Falla en presión hidráulica en freno Perfiladores
   DF_021 : BOOL ;	//Falla de excursión en Ajuste de ancho de Perfiladores
   DF_022 : BOOL ;	//Falla de excursión en Ajuste de ancho de Formado
   DF_023 : BOOL ;	//Falla de seguridad en Perímetro
   DF_024 : BOOL ;	//Reserva
   DF_025 : BOOL ;	//Falla alimentación de Entradas
   DF_026 : BOOL ;	//Falla de seguridad
   DF_027 : BOOL ;	//Falla presión de Aire
   DF_028 : BOOL ;	//Falla Temperatura Grupo Hidráulico
   DF_029 : BOOL ;	//Falla Seguridad Barrera en Descargador
   DF_030 : BOOL ;	//Falla Cubierta de Perfilador
   DF_031 : BOOL ;	//Falla de Atasco de pieza en Perfilador
   DF_032 : BOOL ;	//Reserva
   DF_033 : BOOL ;	//Falla avance de pinza en Plegadora
   DF_034 : BOOL ;	//Falla al bajar pinza en Plegadora
   DF_035 : BOOL ;	//Falla al abrir pinza en Plegadora
   DF_036 : BOOL ;	//Falla activar alineación eje X (ANULADA)
   DF_037 : BOOL ;	//Falla activar alineación eje Y (ANULADA)
   DF_038 : BOOL ;	//Falla Subir Cepillos (ANULADA)
   DF_039 : BOOL ;	//Reserva
   DF_040 : BOOL ;	//Reserva
   DF_041 : BOOL ;	//Falla retroceso de pinza en Plegadora
   DF_042 : BOOL ;	//Falla al subir pinza en Plegadora
   DF_043 : BOOL ;	//Falla al cerrar pinza en Plegadora
   DF_044 : BOOL ;	//Falla desactivar alineación eje X (ANULADA)
   DF_045 : BOOL ;	//Falla desactivar alineación eje Y (ANULADA)
   DF_046 : BOOL ;	//Falla Bajar Cepillos (ANULADA)
   DF_047 : BOOL ;	//Reserva
   DF_048 : BOOL ;	//Reserva
   DF_049 : BOOL ;	//Falla Subir Fijaciones Plegador 1
   DF_050 : BOOL ;	//Falla Subir Plegador 1
   DF_051 : BOOL ;	//Falla Subir Prensa Plegador 1
   DF_052 : BOOL ;	//Falla Subir Extensión 1 Prensa Plegador 1
   DF_053 : BOOL ;	//Falla Subir Fijaciones Plegador 2
   DF_054 : BOOL ;	//Falla Subir Plegador 2
   DF_055 : BOOL ;	//Falla Subir Prensa Plegador 2
   DF_056 : BOOL ;	//Falla Subir Extensión 1 Prensa Plegador 2
   DF_057 : BOOL ;	//Falla Bajar Fijaciones Plegador 1
   DF_058 : BOOL ;	//Falla Bajar Plegador 1
   DF_059 : BOOL ;	//Falla Bajar Prensa Plegador 1
   DF_060 : BOOL ;	//Falla Bajar Extensión 1 Prensa Plegador 1
   DF_061 : BOOL ;	//Falla Bajar Fijaciones Plegador 2
   DF_062 : BOOL ;	//Falla Bajar Plegador 2
   DF_063 : BOOL ;	//Falla Bajar Prensa Plegador 2
   DF_064 : BOOL ;	//Falla Bajar Extensión 1 Prensa Plegador 2
   DF_065 : BOOL ;	//Falla Avance Transporte de Araña
   DF_066 : BOOL ;	//Fallas Subir Araña
   DF_067 : BOOL ;	//Fallas Bajar Araña Pistón 2
   DF_068 : BOOL ;	//Fallas Subir Araña Pistón 2
   DF_069 : BOOL ;	//Reserva
   DF_070 : BOOL ;	//Reserva
   DF_071 : BOOL ;	//Reserva
   DF_072 : BOOL ;	//Reserva
   DF_073 : BOOL ;	//Falla Retroceso Transporte de Araña
   DF_074 : BOOL ;	//Fallas Bajar Araña
   DF_075 : BOOL ;	//Reserva
   DF_076 : BOOL ;	//Reserva
   DF_077 : BOOL ;	//Falla Subir Extensión 2 Prensa Plegador 1
   DF_078 : BOOL ;	//Falla Subir Extensión 2 Prensa Plegador 2
   DF_079 : BOOL ;	//Falla Bajar Extensión 2 Prensa Plegador 1
   DF_080 : BOOL ;	//Falla Bajar Extensión 2 Prensa Plegador 2
   DF_081 : BOOL ;	//Falla Avance Ajuste de Formado (ANULADA)
   DF_082 : BOOL ;	//Falla Subir Bloqueo de avance Formador
   DF_083 : BOOL ;	//Falla Abrir Pinza
   DF_084 : BOOL ;	//Reserva
   DF_085 : BOOL ;	//Falla Retroceso Ajuste de Formado (ANULADA)
   DF_086 : BOOL ;	//Falla Bajar Bloqueo de avance Formador
   DF_087 : BOOL ;	//Falla Cerrar Pinza
   DF_088 : BOOL ;	//Reserva
   DF_089 : BOOL ;	//Falla ON Martillo de Herramienta 1 de Formado
   DF_090 : BOOL ;	//Falla ON Matriz de Herramienta 1 de Formad
   DF_091 : BOOL ;	//Falla ON Martillo de Herramienta 2 de Formado
   DF_092 : BOOL ;	//Falla ON Matriz de Herramienta 2 de Formado
   DF_093 : BOOL ;	//Falla Bloqueo de Herramientas de Formado
   DF_094 : BOOL ;	//Fallas Avanzar Descargador
   DF_095 : BOOL ;	//Falla Avance Intercambiador de Almacenes
   DF_096 : BOOL ;	//Reserva
   DF_097 : BOOL ;	//Falla OFF Martillo de Herramienta 1 de Formado
   DF_098 : BOOL ;	//Falla OFF Matriz de Herramienta 1 de Formado
   DF_099 : BOOL ;	//Falla OFF Martillo de Herramienta 2 de Formado
   DF_100 : BOOL ;	//Falla OFF Matriz de Herramienta 2 de Formado
   DF_101 : BOOL ;	//Falla Desbloqueo de Herramientas de Formado
   DF_102 : BOOL ;	//Falla Retroceder Descargador
   DF_103 : BOOL ;	//Falla Retroceso Intercambiador de Almacenes
   DF_104 : BOOL ;	//Reserva
   DF_105 : BOOL ;	//Reserva
   DF_106 : BOOL ;	//Reserva
   DF_107 : BOOL ;	//Reserva
   DF_108 : BOOL ;	//Reserva
   DF_109 : BOOL ;	//Reserva
   DF_110 : BOOL ;	//Reserva
   DF_111 : BOOL ;	//Reserva
   DF_112 : BOOL ;	//Reserva
   DF_113 : BOOL ;	//Reserva
   DF_114 : BOOL ;	//Reserva
   DF_115 : BOOL ;	//Reserva
   DF_116 : BOOL ;	//Inconsistencia de Presencia de pieza en Transporte de Rolos
   DF_117 : BOOL ;	//Reserva
   DF_118 : BOOL ;	//Reserva
   DF_119 : BOOL ;	//Reserva
   DF_120 : BOOL ;	//Reserva
   DF_121 : BOOL ;	//Inconsistencia de Presencia de pieza en en Descargador
   DB_VAR1 : ARRAY  [1 .. 7 ] OF //Variable Temporal
   INT  := 0;
   DEF01 : INT ;	//IMAGE DEFAUT DBW 50
   DEF02 : INT ;	//IMAGE DEFAUT DBW 52
   DEF03 : INT ;	//IMAGE DEFAUT DBW 54
   DEF04 : INT ;	//IMAGE DEFAUT DBW 56
   DEF05 : INT ;	//IMAGE DEFAUT DBW 58
   DEF06 : INT ;	//IMAGE DEFAUT DBW 60
   DEF07 : INT ;	//IMAGE DEFAUT DBW 62
   DEF08 : INT ;	//IMAGE DEFAUT DBW 64
   DEF09 : INT ;	//IMAGE DEFAUT DBW
   DEF10 : INT ;	//IMAGE DEFAUT DBW 50
   COD1_VAL : DINT ;	//Encoder Perfilador 1 : Valor 1/10 mm
   COD1_CONS : DINT ;	//Encoder Perfilador 1 : Consigna Posición 1/10 mm
   COD1_ARRET : DINT ;	//Encoder Perfilador 1 : Parar 1/10 mm
   COD1_TARGET : DINT ;	//Encoder Perfilador 1 : Ventana 1/10 mm
   COD1_INIT : DINT ;	//Encoder Perfilador 1 : Consigna Inicial  1/10 mm
   COD1_COEF : REAL  := 1.000000e+000;	//Encoder Perfilador 1 : Coeficiente Corrección
   COD1_RES : ARRAY  [1 .. 2 ] OF //Variable temporal
   INT  := 0;
   COD1_CMD : BOOL ;	//Encoder Perfilador 1 : Inicio
   COD1_MOP : BOOL ;	//Encoder Perfilador 1 : Ajuste en Operación
   COD1_MPO_AV : BOOL ;	//Encoder Perfilador 1 : MOP Avance
   COD1_MPO_RC : BOOL ;	//Encoder Perfilador 1 : MOP Retroceso
   COD1_MPO_OK : BOOL ;	//Encoder Perfilador 1 : MOP OK
   COD2_VAL : DINT ;	//Encoder Formador 2 : Valor 1/10 mm
   COD2_CONS : DINT ;	//Encoder Formador 2 : Consigna Posición  1/10 mm
   COD2_ARRET : DINT ;	//Encoder Formador 2 : Parar 1/10 mm
   COD2_TARGET : DINT ;	//Encoder Formador 2 : Ventana 1/10 mm
   COD2_INIT : DINT ;	//Encoder Formador 2 : Consigna Inicial  1/10 mm
   COD2_COEF : REAL  := 1.000000e+000;	//Encoder Formador 2 : Coeficiente Corrección
   COD2_RES : ARRAY  [1 .. 2 ] OF //Variable temporales
   INT  := 0;
   COD2_CMD : BOOL ;	//Encoder Formador 2 : Inicio
   COD2_MOP : BOOL ;	//Encoder Perfilador 2 : Ajuste en Operación
   COD2_MPO_AV : BOOL ;	//Encoder Perfilador 2 : MOP Avance
   COD2_MPO_RC : BOOL ;	//Encoder Perfilador 2 : MOP Retroceso
   COD2_MPO_OK : BOOL ;	//Encoder Perfilador 2 : MOP OK
   COD_RES : ARRAY  [1 .. 20 ] OF //Variable temporal
   INT  := 0;
   PL1_POS_ENCODER : DINT ;	//Encoder Plegador 1 : Valor ( x 0.1 mm)
   PL1_POS_CONSIGNA : DINT ;	//Encoder Plegador 1 : Consigna Posición  ( x 0.1 mm)
   PL1_POS_CONSIGNA_INICIO : DINT ;	//Encoder Plegador 1 : Consigna Inicial  ( x 0.1 mm)
   PL1_COD_COEF : REAL  := 1.000000e+000;	//Encoder Plegador 1 : Coeficiente Corrección
   PL1_VEL_AUTO : INT  := 10;	//Encoder Plegador 1 : Velocidad Automática %
   PL1_COD1_RES1 : ARRAY  [1 .. 15 ] OF //Variable temporal
   INT  := 0;
   PL1_COD_CMD : BOOL ;	//Encoder Plegador 2 : Inicio
   PL2_POS_ENCODER : DINT ;	//Encoder Plegador 2 : ( x 0.1 mm)
   PL2_POS_CONSIGNA : DINT ;	//Encoder Plegador 2 : Consigna Posición  ( x 0.1 mm)
   PL2_POS_CONSIGNA_INICIO : DINT ;	//Encoder Plegador 2 : Consigna Inicial  ( x 0.1 mm)
   PL2_COD_COEF : REAL  := 1.000000e+000;	//Encoder Plegador 2 : Coeficiente Corrección
   PL2_VEL_AUTO : INT  := 10;	//Encoder Plegador 2 : Velocidad Automática %
   PL2_COD_RES : ARRAY  [1 .. 15 ] OF //Variable temporal
   INT  := 0;
   PL2_COD_CMD : BOOL ;	//Encoder Plegador 2 : Inicio
   PI_POS_ENCODER : DINT ;	//Encóder Pinza : ( x 0.1 mm)
   PI_POS_CONSIGNA : DINT ;	//Encóder Pinza : Consigna Posición ( x 0.1 mm)
   PI_POS_CONSIGNA_INICIO : DINT ;	//Encóder Pinza : Consigna Inicial ( x 0.1 mm)
   PI_COD_COEF : REAL  := 1.000000e+000;	//Encóder Pinza : Coeficiente Corrección
   PI_VEL_ATUO : INT  := 10;	//Encóder Pinza : Velocidad Automática %
   PI_Dist_Inicio_H1 : DINT  := L#112500;	//Encóder Pinza : Distancia Posición Inicial a Herramienta 1
   PI_Dist_Inicio_Tenaza : DINT  := L#218000;	//Encóder Pinza : Distancia Posición Inicial a Tenaza Plegadora
   PI_COD1_RES : ARRAY  [1 .. 11 ] OF //Variable temporal
   INT  := 0;
   PI_COD_CMD : BOOL ;	//Encóder Plegador 2 : Inicio
   RESERVE : ARRAY  [1 .. 11 ] OF //Variable temporal
   INT  := 0;
   M1_P_CPT : INT ;	//Almacén 1 Preselección contador de piezas
   M1_V_CPT : INT ;	//Almacén 1 contador de piezas
   M2_P_CPT : INT ;	//Almacén 2 Preselección contador de piezas
   M2_V_CPT : INT ;	//Almacén 2 contador de piezas
   M1T_XCPT : BOOL ;	//Almacén 1 Entrega Pieza
   M1_AP_PH : BOOL ;	//Almacén 1 Autorizado
   M1T : BYTE ;	//Almacén 1
   M2_XCPT : BOOL ;	//Almacén 2 Entrega Pieza
   M2_AP_PH : BOOL ;	//Almacén 2 Autorizado
   M2T : BYTE ;	//Almacén 2
   PHT : INT ;	//Almacén 1 Motor trabajando
   C1T : INT ;	//Almacén 1 Motor trabajando
   PFT : INT ;	//Almacén 2 Motor trabajando
   C2T : INT ;	//Almacén 2 Motor trabajando
   Pinza_Recepcion : BOOL ;	//Pinza en posición Recepción
   Pinza_E1H1 : BOOL ;	//Ultimo Posicionamiento E1H1 (F1)
   Pinza_E1H2 : BOOL ;	//Ultimo Posicionamiento E1H2 (F2)
   Pinza_E2H1 : BOOL ;	//Ultimo Posicionamiento E2H1 (F3)
   Pinza_E2H2 : BOOL ;	//Ultimo Posicionamiento E2H2 (F4)
   Pinza_Entrega : BOOL ;	//Ultimo Posicionamiento Entrega
  END_STRUCT ;	
BEGIN
   MODE := 3;
   RC1 := 2;
   RC2 := 9;
   COD1_COEF := 1.000000e+00;
   COD2_COEF := 1.000000e+00;
   PL1_COD_COEF := 1.000000e+00;
   PL1_VEL_AUTO := 10;
   PL2_COD_COEF := 1.000000e+00;
   PL2_VEL_AUTO := 10;
   PI_COD_COEF := 1.000000e+00;
   PI_VEL_ATUO := 10;
   PI_Dist_Inicio_H1 := L#112500;
   PI_Dist_Inicio_Tenaza := L#218000;
END_DATA_BLOCK

DATA_BLOCK "Posiciones Plegador 2"	// DB 54
VERSION : 0.1
  STRUCT
   ChapaCompleta : DINT ;
   STAT1 : DINT ;
   Espera : DINT ;
   Recepcion : DINT ;
   Plegado1 : DINT ;
   Plegado2 : DINT ;
   Entrega : DINT ;
   STAT7 : DINT ;
   STAT8 : DINT ;
   STAT9 : DINT ;
   STAT10 : DINT ;
   STAT11 : DINT ;
   STAT12 : DINT ;
  END_STRUCT ;	
BEGIN
END_DATA_BLOCK

DATA_BLOCK "Posiciones Plegador 1"	// DB 55
VERSION : 0.1
  STRUCT
   ChapaCompleta : DINT ;
   STAT1 : DINT ;
   Espera : DINT ;
   Recepcion : DINT ;
   Plegado1 : DINT ;
   Plegado2 : DINT ;
   Entrega : DINT ;
   STAT7 : DINT ;
   STAT8 : DINT ;
   STAT9 : DINT ;
   STAT10 : DINT ;
   STAT11 : DINT ;
   STAT12 : DINT ;
  END_STRUCT ;	
BEGIN
   ChapaCompleta := L#348380;
   STAT1 := L#348380;
   Espera := L#30000;
   Recepcion := L#118910;
   Plegado1 := L#172309;
   Plegado2 := L#30200;
   Entrega := L#27000;
END_DATA_BLOCK

DATA_BLOCK "Posiciones Plegadores 00"	// DB 56
AUTHOR : EMR
NAME : eProC
VERSION : 0.1
  STRUCT
   ChapaCompleta : DINT  := L#30000;
   STAT1 : DINT  := L#30000;
   Espera : DINT  := L#30000;
   Recepcion : DINT  := L#30000;
   Plegado1 : DINT  := L#30000;
   Plegado2 : DINT  := L#30000;
   Entrega : DINT  := L#30000;
   STAT7 : DINT  := L#30000;
   STAT8 : DINT  := L#30000;
   STAT9 : DINT  := L#30000;
   STAT10 : DINT  := L#30000;
   STAT11 : DINT  := L#30000;
   STAT12 : DINT  := L#30000;
  END_STRUCT ;	
BEGIN
   ChapaCompleta := L#30000;
   STAT1 := L#30000;
   Espera := L#30000;
   Recepcion := L#30000;
   Plegado1 := L#30000;
   Plegado2 := L#30000;
   Entrega := L#30000;
   STAT7 := L#30000;
   STAT8 := L#30000;
   STAT9 := L#30000;
   STAT10 := L#30000;
   STAT11 := L#30000;
   STAT12 := L#30000;
END_DATA_BLOCK

DATA_BLOCK "Posiciones Pleg. 1 Ant"	// DB 57
VERSION : 0.1
  STRUCT
   ChapaCompleta : DINT ;
   STAT1 : DINT ;
   Espera : DINT ;
   Recepcion : DINT ;
   Plegado1 : DINT ;
   Plegado2 : DINT ;
   Entrega : DINT ;
   STAT7 : DINT ;
   STAT8 : DINT ;
   STAT9 : DINT ;
   STAT10 : DINT ;
   STAT11 : DINT ;
   STAT12 : DINT ;
  END_STRUCT ;	
BEGIN
   ChapaCompleta := L#348380;
   STAT1 := L#348380;
   Espera := L#30000;
   Recepcion := L#118910;
   Plegado1 := L#172309;
   Plegado2 := L#30200;
   Entrega := L#27000;
END_DATA_BLOCK

DATA_BLOCK "Posiciones Pleg. 2 Ant"	// DB 58
VERSION : 0.1
  STRUCT
   ChapaCompleta : DINT ;
   STAT1 : DINT ;
   Espera : DINT ;
   Recepcion : DINT ;
   Plegado1 : DINT ;
   Plegado2 : DINT ;
   Entrega : DINT ;
   STAT7 : DINT ;
   STAT8 : DINT ;
   STAT9 : DINT ;
   STAT10 : DINT ;
   STAT11 : DINT ;
   STAT12 : DINT ;
  END_STRUCT ;	
BEGIN
END_DATA_BLOCK

ORGANIZATION_BLOCK OB 1
VERSION : 0.1
VAR_TEMP
  OB1_EV_CLASS : BYTE ;	//Bits 0-3 = 1 (Coming event), Bits 4-7 = 1 (Event class 1)
  OB1_SCAN_1 : BYTE ;	//1 (Cold restart scan 1 of OB 1), 3 (Scan 2-n of OB 1)
  OB1_PRIORITY : BYTE ;	//Priority of OB Execution
  OB1_OB_NUMBR : BYTE ;	//1 (Organization block 1, OB1)
  OB1_RESERVED_1 : BYTE ;	//Reserved for system
  OB1_RESERVED_2 : BYTE ;	//Reserved for system
  OB1_PREV_CYCLE : INT ;	//Cycle time of previous OB1 scan (milliseconds)
  OB1_MIN_CYCLE : INT ;	//Minimum cycle time of OB1 (milliseconds)
  OB1_MAX_CYCLE : INT ;	//Maximum cycle time of OB1 (milliseconds)
  OB1_DATE_TIME : DATE_AND_TIME ;	//Date and time OB1 started
END_VAR
BEGIN
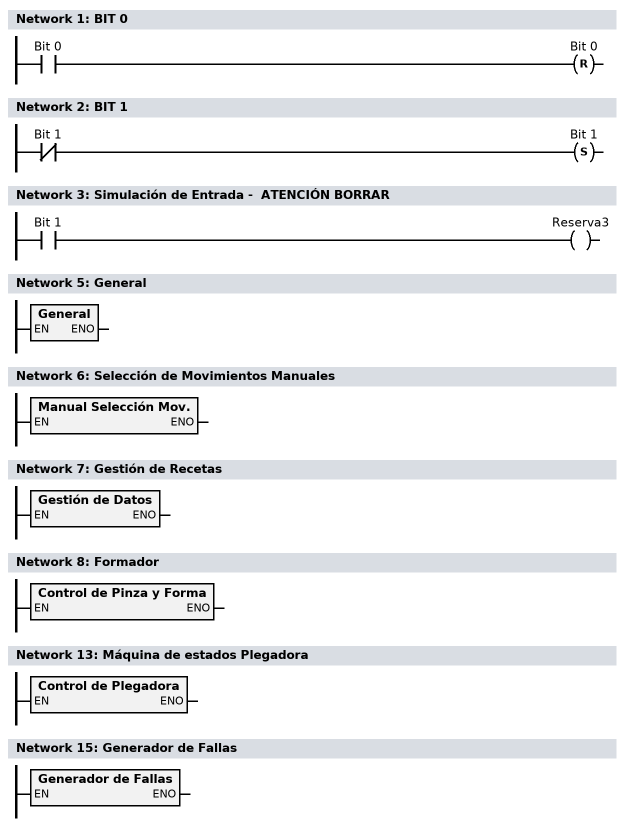
NETWORK
TITLE = BIT 0
      A     "Bit 0";
      R     "Bit 0";
NETWORK
TITLE = BIT 1
      AN    "Bit 1";
      S     "Bit 1";
NETWORK
TITLE = Simulación de Entrada -  ATENCIÓN BORRAR
      A     "Bit 1";
      =     "Reserva3";
NETWORK
TITLE =
NETWORK
TITLE = General
      CALL  "General";
      NOP   0;
NETWORK
TITLE = Selección de Movimientos Manuales
      CALL  "Manual Selección Mov.";
      NOP   0;
NETWORK
TITLE = Gestión de Recetas
      CALL  "Gestión de Datos";
      NOP   0;
NETWORK
TITLE = Formador
      CALL  "Control de Pinza y Forma";
      NOP   0;
NETWORK
TITLE = Almacenes
      UC    "Almacenes";
NETWORK
TITLE = Transportes
      UC    "Transportes";
NETWORK
TITLE = Perfilador
      UC    "Perfilador";
NETWORK
TITLE = Araña
      UC    "Araña";
NETWORK
TITLE = Máquina de estados Plegadora
      CALL  "Control de Plegadora";
      NOP   0;
NETWORK
TITLE = Descarga
      UC    "Descarga";
NETWORK
TITLE = Generador de Fallas
      CALL  "Generador de Fallas";
      NOP   0;
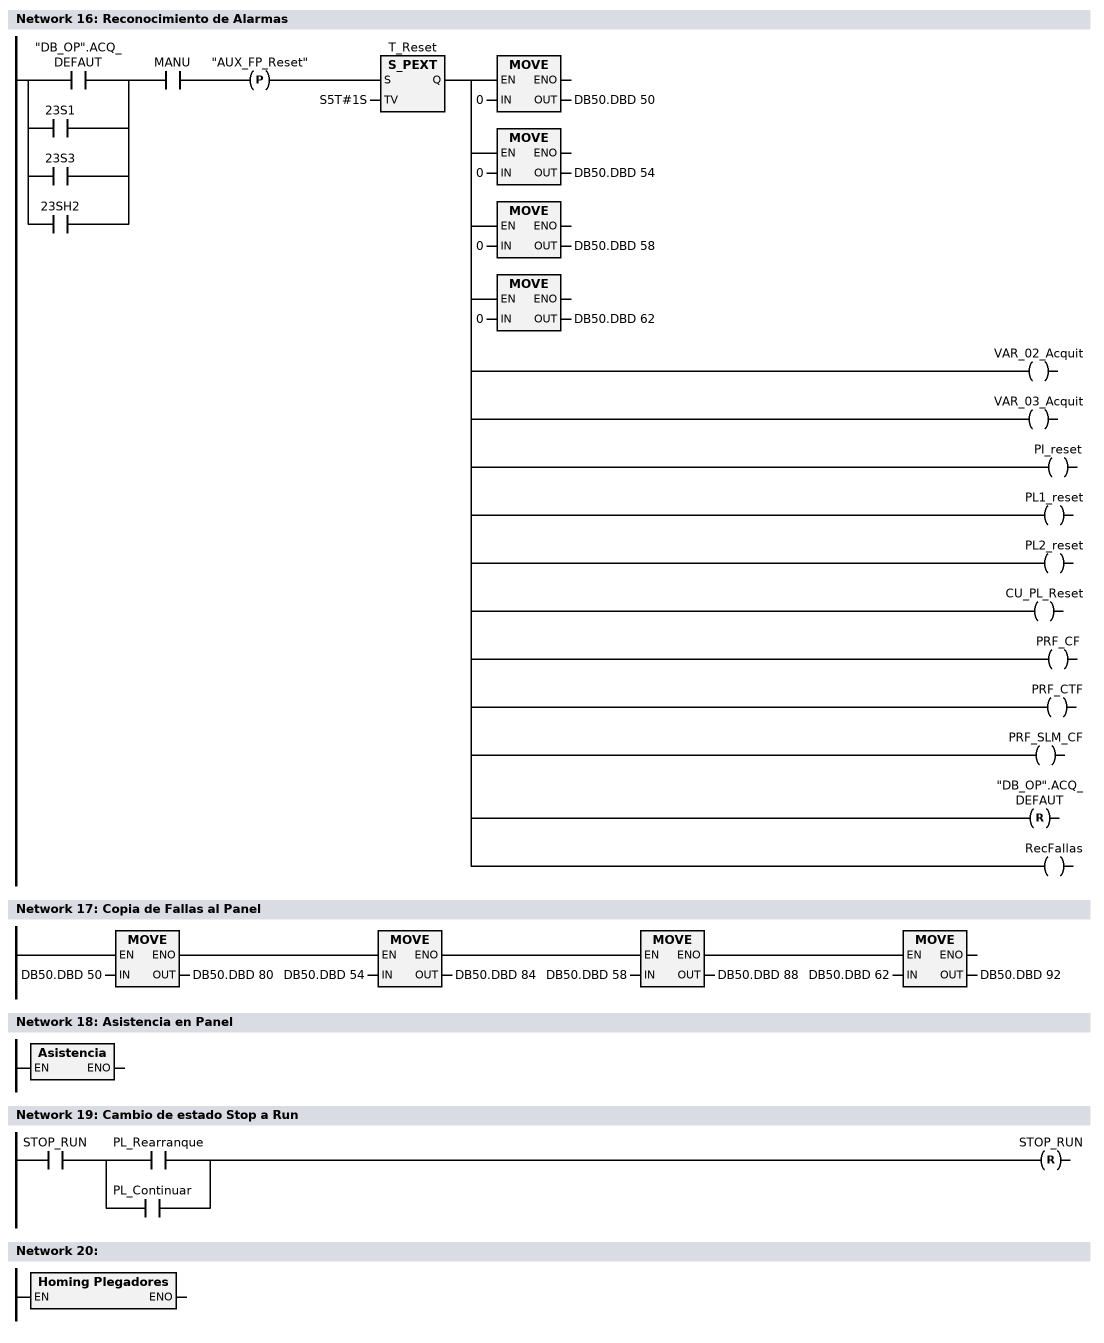
NETWORK
TITLE = Reconocimiento de Alarmas
      A(;
      O     "DB_OP".ACQ_DEFAUT;
      O     "23S1";
      O     "23S3";
      O     "23SH2";
      );
      A     "MANU";
      FP    "AUX_FP_Reset";
      L     S5T#1S;
      SE    "T_Reset";
      NOP   0;
      NOP   0;
      NOP   0;
      A     "T_Reset";
      =     L 20.0;
      A     L 20.0;
      JNB   _001;
      L     0;
      T     DB50.DBD 50;
_001: NOP   0;
      A     L 20.0;
      JNB   _002;
      L     0;
      T     DB50.DBD 54;
_002: NOP   0;
      A     L 20.0;
      JNB   _003;
      L     0;
      T     DB50.DBD 58;
_003: NOP   0;
      A     L 20.0;
      JNB   _004;
      L     0;
      T     DB50.DBD 62;
_004: NOP   0;
      A     L 20.0;
      BLD   102;
      =     "VAR_02_Acquit";
      A     L 20.0;
      BLD   102;
      =     "VAR_03_Acquit";
      A     L 20.0;
      BLD   102;
      =     "PI_reset";
      A     L 20.0;
      BLD   102;
      =     "PL1_reset";
      A     L 20.0;
      BLD   102;
      =     "PL2_reset";
      A     L 20.0;
      BLD   102;
      =     "CU_PL_Reset";
      A     L 20.0;
      BLD   102;
      =     "PRF_CF";
      A     L 20.0;
      BLD   102;
      =     "PRF_CTF";
      A     L 20.0;
      BLD   102;
      =     "PRF_SLM_CF";
      A     L 20.0;
      BLD   102;
      R     "DB_OP".ACQ_DEFAUT;
      A     L 20.0;
      BLD   102;
      =     "RecFallas";
NETWORK
TITLE = Copia de Fallas al Panel
      A(;
      A(;
      A(;
      L     DB50.DBD 50;
      T     DB50.DBD 80;
      SET;
      SAVE;
      CLR;
      A     BR;
      );
      JNB   _005;
      L     DB50.DBD 54;
      T     DB50.DBD 84;
      SET;
      SAVE;
      CLR;
_005: A     BR;
      );
      JNB   _006;
      L     DB50.DBD 58;
      T     DB50.DBD 88;
      SET;
      SAVE;
      CLR;
_006: A     BR;
      );
      JNB   _007;
      L     DB50.DBD 62;
      T     DB50.DBD 92;
_007: NOP   0;
NETWORK
TITLE = Asistencia en Panel
      CALL  "Asistencia";
      NOP   0;
NETWORK
TITLE = Cambio de estado Stop a Run
      A     "STOP_RUN";
      A(;
      O     "PL_Rearranque";
      O     "PL_Continuar";
      );
      R     "STOP_RUN";
NETWORK
TITLE =
      CALL  "Homing Plegadores";
      NOP   0;
END_ORGANIZATION_BLOCK

ORGANIZATION_BLOCK "I/O_FLT1"	// OB 82
VERSION : 0.0
BEGIN
// (block stored without names or comments; labels and parameter names are numbered)
END_ORGANIZATION_BLOCK

ORGANIZATION_BLOCK "RACK_FLT"	// OB 86
VERSION : 0.0
BEGIN
// (block stored without names or comments; labels and parameter names are numbered)
END_ORGANIZATION_BLOCK

ORGANIZATION_BLOCK "COMPLETE RESTART"	// OB 100
TITLE = "Complete Restart"
VERSION : 0.1
VAR_TEMP
  OB100_EV_CLASS : BYTE ;	//16#13, Event class 1, Entering event state, Event logged in diagnostic buffer
  OB100_STRTUP : BYTE ;	//16#81/82/83/84 Method of startup
  OB100_PRIORITY : BYTE ;	//Priority of OB Execution
  OB100_OB_NUMBR : BYTE ;	//100 (Organization block 100, OB100)
  OB100_RESERVED_1 : BYTE ;	//Reserved for system
  OB100_RESERVED_2 : BYTE ;	//Reserved for system
  OB100_STOP : WORD ;	//Event that caused CPU to stop (16#4xxx)
  OB100_STRT_INFO : DWORD ;	//Information on how system started
  OB100_DATE_TIME : DATE_AND_TIME ;	//Date and time OB100 started
END_VAR
BEGIN
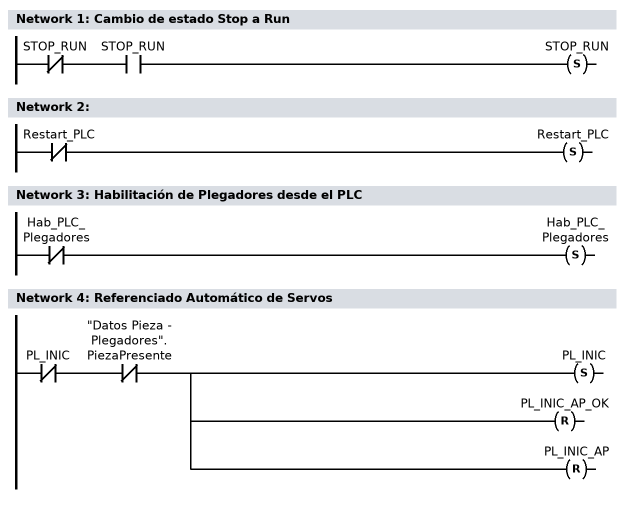
NETWORK
TITLE = Cambio de estado Stop a Run
      AN    "STOP_RUN";
      A     "STOP_RUN";
      S     "STOP_RUN";
NETWORK
TITLE =
      AN    "Restart_PLC";
      S     "Restart_PLC";
NETWORK
TITLE = Habilitación de Plegadores desde el PLC
      AN    "Hab_PLC_Plegadores";
      S     "Hab_PLC_Plegadores";
NETWORK
TITLE = Referenciado Automático de Servos
      AN    "PL_INIC";
      AN    "Datos Pieza - Plegadores".PiezaPresente;
      S     "PL_INIC";
      R     "PL_INIC_AP_OK";
      R     "PL_INIC_AP";
END_ORGANIZATION_BLOCK

ORGANIZATION_BLOCK "PROG_ERR"	// OB 121
VERSION : 0.0
BEGIN
// (block stored without names or comments; labels and parameter names are numbered)
END_ORGANIZATION_BLOCK

ORGANIZATION_BLOCK "MOD_ERR"	// OB 122
TITLE = "Module Access Error"
VERSION : 0.1
VAR_TEMP
  OB122_EV_CLASS : BYTE ;	//16#29, Event class 2, Entering event state, Internal fault event
  OB122_SW_FLT : BYTE ;	//16#XX Software error code
  OB122_PRIORITY : BYTE ;	//Priority of OB Execution
  OB122_OB_NUMBR : BYTE ;	//122 (Organization block 122, OB122)
  OB122_BLK_TYPE : BYTE ;	//16#88/8C/8E Type of block fault occured in
  OB122_MEM_AREA : BYTE ;	//Memory area where access error occured
  OB122_MEM_ADDR : WORD ;	//Memory address where access error occured
  OB122_BLK_NUM : WORD ;	//Block number in which error occured
  OB122_PRG_ADDR : WORD ;	//Program address where error occured
  OB122_DATE_TIME : DATE_AND_TIME ;	//Date and time OB1 started
END_VAR
BEGIN
// (block stored without names or comments; labels and parameter names are numbered)
END_ORGANIZATION_BLOCK
